	PROCESSING:
		CASE THIS^.intersectIterator.iterate(execute := TRUE, object => iteratedObject) OF
		CNM_ReturnTypes.SingleExecutionState.BUSY:
			IF THIS^.getEqualObject(object := iteratedObject, foundObject => intersectObject) THEN
				IF (THIS^.intersectedTree^.insert(intersectObject) <> CNM_ReturnTypes.SingleExecutionResult.ERROR) THEN
					insertOperationsThisCycle := insertOperationsThisCycle + log2(THIS^.intersectedTree^.size);
				ELSE
					cycleManager.proceedWith(ERROR);
					CONTINUE;
				END_IF
			END_IF
			insertOperationsThisCycle := insertOperationsThisCycle + log2(THIS^.size);
		CNM_ReturnTypes.SingleExecutionState.ERROR:
			cycleManager.proceedWith(ERROR);
			CONTINUE;
		CNM_ReturnTypes.SingleExecutionState.SUCCESS:
			THIS^.clear();
			THIS^.root := THIS^.intersectedTree^.root;
			THIS^.size := THIS^.intersectedTree^.size;
			THIS^.intersectedTree^.root := 0;
			THIS^.intersectedTree^.destruct();
			THIS^.intersectedTree := 0;
			THIS^.intersectIterator.destruct();
			THIS^.intersectIterator := 0;
			cycleManager.proceedWith(SUCCESS);
			CONTINUE;
		END_CASE
	
	ERROR:
		THIS^.intersectIterator.destruct();
		THIS^.intersectIterator := 0;
		__DELETE(THIS^.intersectedTree);
		THIS^.intersectedTree := 0;
	END_CASE	
UNTIL
	(insertOperationsThisCycle >= THIS^.maxCycleCompares) OR_ELSE
	(cycleManager.state <> CNM_ReturnTypes.SingleExecutionState.BUSY)
END_REPEAT

intersect := cycleManager.state;
END_METHOD


(*

## Short summary

This method returns the next object in the iteration and returns an execution state.

.. <legal notes>

legal notes
=================
| SPDX-FileCopyrightText: © 2022 ekvip automation GmbH <info@ekvip.de>
| SPDX-License-Identifier: Apache-2.0
| For details check: Apache-2.0_

.. _Apache-2.0: https://www.apache.org/licenses/LICENSE-2.0

.. </legal notes>


**Return:** ``SUCCESS``: if last object from collection was returned,
	``ABORTED``: execute has a falling edge during iterate,
	``BUSY``: When iterate had rising edge on execute and not all objects had been returned yet
	``IDLE``: iterate not in progress, execute is false and iterate reseted 
	
*)

METHOD PROTECTED iterate :CNM_ReturnTypes.SingleExecutionState
VAR_INPUT
	execute					:BOOL;
END_VAR
VAR_OUTPUT
	object					:CNM_AbstractObject.IObject;
END_VAR
VAR_INST
	currentNode				:CNM_CollectionInterfaces.IBinaryTreeNode;
	stacktop				:__XWORD := 0;
	cycleManager	:CNM_CycleManager.SimpleCycleManager;
	lastTreeVersion :__XWORD;
END_VAR
VAR 
	stacksize 				:UDINT;
END_VAR
VAR CONSTANT 
	INIT :DINT := CNM_ReturnTypes.DefaultSteps.STEP.INIT;
	ITERATING :DINT := INIT + 1;
	SUCCESS :DINT := CNM_ReturnTypes.DefaultSteps.STEP.SUCCESS;
	ERROR :DINT := CNM_ReturnTypes.DefaultSteps.STEP.ERROR;
	OBJECT_NOT_REFERENCED	:__XWORD := 0;
END_VAR
cycleManager(execute := execute);
CASE cycleManager.step.current OF
INIT:
	cycleManager.configuration.sequence.requireSuccessStep := FALSE;
	stacksize := THIS^.treeHeight;
	object := OBJECT_NOT_REFERENCED;
	lastTreeVersion := THIS^.changesToCollection;
	__DELETE(THIS^.nodestack);
	stacktop := 0;
	THIS^.nodestack := __NEW(__XWORD, stacksize);
	currentNode := THIS^.getSmallestNode(startNode:=THIS^.rootNode,nodebuffer := THIS^.nodestack,bufferindex := stacktop);
	IF THIS^.isObjectValid(currentNode) THEN
		object := currentNode.object;
		THIS^.getInorderSuccessor(
          nodebuffer := THIS^.nodestack, 
          bufferindex := stacktop, 
          successor => currentNode
        );
	END_IF
	cycleManager.proceedWith(
		step := SEL((THIS^.size > 0), SUCCESS, ITERATING)
	);
	
ITERATING:
	IF THIS^.changesToCollection <> lastTreeVersion THEN
		cycleManager.proceedWith(ERROR);
		iterate := CNM_ReturnTypes.SingleExecutionState.ERROR;
		RETURN;
	END_IF
	IF THIS^.isObjectValid(currentNode) THEN
		object := currentNode.object;
		THIS^.getInorderSuccessor(
          nodebuffer := THIS^.nodestack, 
          bufferindex := stacktop, 
          successor => currentNode
        );
	ELSE
		__DELETE(THIS^.nodestack);
		cycleManager.proceedWith(SUCCESS);
	END_IF
END_CASE

iterate := cycleManager.state;
END_METHOD

(*

## Short summary

This property defines the maximum amount of compares that should be done per Cycle. Is optional as default should be set by class.
Passing zero resets to class specific default.

.. <legal notes>

legal notes
=================
| SPDX-FileCopyrightText: © 2022 ekvip automation GmbH <info@ekvip.de>
| SPDX-License-Identifier: Apache-2.0
| For details check: Apache-2.0_

.. _Apache-2.0: https://www.apache.org/licenses/LICENSE-2.0

.. </legal notes>

*)

PROPERTY maxCycleCompares : UDINT
GET
maxCycleCompares := THIS^.upperCompareBound;
END_GET
SET
THIS^.upperCompareBound := SEL(
	maxCycleCompares = 0,
	maxCycleCompares,
	GeneralParameters.DEFAULT_OPERATIONS_PER_CYCLE
);
END_SET
END_PROPERTY

(*

## Short summary

overwrites the content of this set with the union of this set and the given set
Set union: Combination of all elements from two sets.

**Example:**
Set A = {2, 3, 1, 4}
Set B = {3, 5, 6, 4}

Union of A and B: {1, 2, 3, 4, 5, 6}

.. <legal notes>

legal notes
=================
| SPDX-FileCopyrightText: © 2022 ekvip automation GmbH <info@ekvip.de>
| SPDX-License-Identifier: Apache-2.0
| For details check: Apache-2.0_

.. _Apache-2.0: https://www.apache.org/licenses/LICENSE-2.0

.. </legal notes>


**Return:** ``SUCCESS``: if merge completed, 
	``ABORTED``: execute has a falling edge during merge,
	``BUSY``: merge is in Progress
	``ERROR``: the passed collection where not valid / contained invalid Elements
	``IDLE``: Currently no merge in progress

*)

METHOD INTERNAL merge :CNM_ReturnTypes.SingleExecutionState
VAR_INPUT
	(*foreign set to merge with*)
	set :CNM_CollectionInterfaces.ISet;
	(*If merge should be processed*)
	execute		:BOOL;
END_VAR
VAR
	object		 	:CNM_AbstractObject.IObject;
	iterateState	:CNM_ReturnTypes.SingleExecutionState;
END_VAR
merge := THIS^.insertCollection(
	collection := set,
	execute := execute);
END_METHOD

(*

## Short summary

recursiv insert function, tries to insert in the Tree and if not on right position call itself again on a subtree, on way out of recursin (re)balance tree

.. <legal notes>

legal notes
=================
| SPDX-FileCopyrightText: © 2022 ekvip automation GmbH <info@ekvip.de>
| SPDX-License-Identifier: Apache-2.0
| For details check: Apache-2.0_

.. _Apache-2.0: https://www.apache.org/licenses/LICENSE-2.0

.. </legal notes>


**Return:** the node that is the new root of the subtree for that the recursiv method is called

*)

METHOD PROTECTED recursivInsert :CNM_CollectionInterfaces.IBalancedBinarySearchTreeNode
VAR_INPUT
	(*the object that shoul be inserted*)
	object 						:CNM_AbstractObject.IObject;
	(*the root of the tree we try to insert in*)
	elem 						:CNM_CollectionInterfaces.IBalancedBinarySearchTreeNode;
END_VAR
VAR_IN_OUT
	(*is changed to false when insert was successful*)
	heightNotChanged 			:BOOL;
END_VAR
VAR 
	rightChild 					:CNM_CollectionInterfaces.IBalancedBinarySearchTreeNode;
	binaryRightChild 			:CNM_CollectionInterfaces.IBinaryTreeNode;
	binaryLeftChild 			:CNM_CollectionInterfaces.IBinaryTreeNode;
	leftChild		  			:CNM_CollectionInterfaces.IBalancedBinarySearchTreeNode;
END_VAR
VAR_OUTPUT
	(*SUCCESS if node could be inserted, ERROR if object already in the tree, ABORTED if object was null or empty node found*)
	insertResult 				:CNM_ReturnTypes.SingleExecutionResult;
END_VAR
VAR CONSTANT
	OBJECT_IS_NOT_REFERENCED	:__XWORD := 0; 
END_VAR
IF THIS^.isObjectNull(elem) AND NOT THIS^.isObjectNull(object) THEN
	IF (THIS^.collectionFactory.getNewBBSTreeNode(object := object, node => recursivInsert) <> CNM_ReturnTypes.SingleExecutionResult.SUCCESS) THEN
		insertResult := CNM_ReturnTypes.SingleExecutionResult.ERROR;
	ELSE
		insertResult := CNM_ReturnTypes.SingleExecutionResult.SUCCESS;
	END_IF
	RETURN;
ELSIF  THIS^.isObjectNull(object) OR_ELSE THIS^.isObjectNull(elem.object) THEN
	insertResult := CNM_ReturnTypes.SingleExecutionResult.ABORTED;
	RETURN;
END_IF
	

CASE THIS^.compareNodes(object, elem.object) OF
 	CNM_ReturnTypes.ComparationResult.EQUAL:
		recursivInsert := elem;
		insertResult := CNM_ReturnTypes.SingleExecutionResult.ABORTED;
		RETURN;
 	CNM_ReturnTypes.ComparationResult.SMALLER: 
		IF (THIS^.isObjectNull(elem.leftChild)) THEN
			IF (THIS^.collectionFactory.getNewBBSTreeNode(object := object, node => leftChild) = CNM_ReturnTypes.SingleExecutionResult.SUCCESS) THEN
				__QUERYINTERFACE(leftChild, binaryLeftChild);
				elem.leftChild := binaryLeftChild;
				heightNotChanged := FALSE;
				insertResult := CNM_ReturnTypes.SingleExecutionResult.SUCCESS;
			ELSE
				insertResult := CNM_ReturnTypes.SingleExecutionResult.ERROR;
			END_IF
		ELSE
			__QUERYINTERFACE(elem.leftChild, leftChild);
			leftChild := THIS^.recursivInsert(object := object, elem := leftChild, heightNotChanged := heightNotChanged, insertResult => insertResult);	
			__QUERYINTERFACE(leftChild,binaryLeftChild);
			elem.leftChild := binaryLeftChild;
		END_IF
		recursivInsert := THIS^.checkRightRotation(elem:=elem,heightNotChanged:=heightNotChanged, removing := FALSE);
		RETURN;
	CNM_ReturnTypes.ComparationResult.Greater:
		IF THIS^.isObjectNull(elem.rightChild) THEN 
			IF (THIS^.collectionFactory.getNewBBSTreeNode(object := object, node => rightChild) = CNM_ReturnTypes.SingleExecutionResult.SUCCESS) THEN
				__QUERYINTERFACE(rightChild,binaryRightChild);
				elem.rightChild := binaryRightChild;
				heightNotChanged := FALSE;
				insertResult := CNM_ReturnTypes.SingleExecutionResult.SUCCESS;
			ELSE
				insertResult := CNM_ReturnTypes.SingleExecutionResult.ERROR;
			END_IF
		ELSE
			__QUERYINTERFACE(elem.rightChild,rightChild);
			rightChild := THIS^.recursivInsert(object:=object,elem:=rightChild,heightNotChanged:=heightNotChanged,insertResult=>insertResult);
			__QUERYINTERFACE(rightChild,binaryRightChild);
			elem.rightChild := binaryRightChild;	
		END_IF
		recursivInsert := THIS^.checkLeftRotation(elem:=elem,heightNotChanged:=heightNotChanged,removing := FALSE);
		RETURN;
END_CASE;
END_METHOD

(*

## Short summary

recursiv remove an element tries to remove element from tree, if not possible calls itself on subtree, on way out of recursin (re)balance tree

.. <legal notes>

legal notes
=================
| SPDX-FileCopyrightText: © 2022 ekvip automation GmbH <info@ekvip.de>
| SPDX-License-Identifier: Apache-2.0
| For details check: Apache-2.0_

.. _Apache-2.0: https://www.apache.org/licenses/LICENSE-2.0

.. </legal notes>


**Return:** the node that is the new root of the subtree for that the recursiv method is called

*)

METHOD PROTECTED recursivRemove :CNM_CollectionInterfaces.IBalancedBinarySearchTreeNode
VAR_INPUT
	(*The object that should be removed*)
	object 						:CNM_AbstractObject.IObject;
	(*The root of the tree we try to delete the object from *)
	elem 						:CNM_CollectionInterfaces.IBalancedBinarySearchTreeNode;
END_VAR
VAR_IN_OUT
	(*changed to false when node is removed*)
	heightNotChanged 			:BOOL;
END_VAR
VAR 
	leftChild					:CNM_CollectionInterfaces.IBalancedBinarySearchTreeNode;
	binaryLeftChild 			:CNM_CollectionInterfaces.IBinaryTreeNode;
	binaryRightChild 			:CNM_CollectionInterfaces.IBinaryTreeNode;
	rightChild 					:CNM_CollectionInterfaces.IBalancedBinarySearchTreeNode;
	testrightChild 				:CNM_CollectionInterfaces.IBinaryTreeNode;
END_VAR
VAR_OUTPUT
	(*SUCCESS, if remove was successful*)
	removeResult 				:CNM_ReturnTypes.SingleExecutionResult;
END_VAR
VAR CONSTANT
	OBJECT_IS_NOT_REFERENCED	:__XWORD := 0;
END_VAR
IF THIS^.isObjectNull(elem) THEN
	recursivRemove := OBJECT_IS_NOT_REFERENCED;
	removeResult := CNM_ReturnTypes.SingleExecutionResult.ABORTED;
	RETURN;
ELSIF THIS^.isObjectNull(object) OR_ELSE THIS^.isObjectNull(elem.object) THEN
	removeResult := CNM_ReturnTypes.SingleExecutionResult.ERROR;
	RETURN;
END_IF;

CASE THIS^.compareNodes(object,elem.object) OF
	CNM_AbstractObject.CNM_ReturnTypes.ComparationResult.SMALLER:
		__QUERYINTERFACE(elem.leftChild,leftChild);
		leftChild := THIS^.recursivRemove(object:=object,elem:=leftChild, heightNotChanged := heightNotChanged,removeResult=>removeResult);
		__QUERYINTERFACE(leftChild,binaryLeftChild);
		elem.leftChild := binaryLeftChild;
		recursivRemove := checkLeftRotation(elem := elem, heightNotChanged := heightNotChanged,removing := TRUE);
		RETURN;
	CNM_AbstractObject.CNM_ReturnTypes.ComparationResult.GREATER:
		__QUERYINTERFACE(elem.rightChild,rightChild);
		rightChild := THIS^.recursivRemove(object := object, elem := rightChild, heightNotChanged := heightNotChanged,removeResult=>removeResult);
		__QUERYINTERFACE(rightChild,binaryRightChild);
		elem.rightChild := binaryRightChild;
		recursivRemove := checkRightRotation(elem := elem, heightNotChanged := heightNotChanged,removing := TRUE);
		RETURN;
	CNM_AbstractObject.CNM_ReturnTypes.ComparationResult.EQUAL:
		IF THIS^.isObjectNull(elem.leftChild) THEN
			heightNotChanged := FALSE;
			__QUERYINTERFACE(elem.rightChild,recursivRemove);
			
		ELSIF THIS^.isObjectNull(elem.rightChild) THEN
			heightNotChanged:=FALSE;
			__QUERYINTERFACE(elem.leftChild,recursivRemove);
		ELSE
			recursivRemove := searchSuccessor(elem:=elem,heightNotChanged:=heightNotChanged);
			recursivRemove.balance := elem.balance;
			recursivRemove.leftChild := elem.leftChild;
			recursivRemove.rightChild := elem.rightChild;
			recursivRemove := checkRightRotation(elem := recursivRemove,heightNotChanged:=heightNotChanged,removing := TRUE);
		END_IF
		removeResult := CNM_ReturnTypes.SingleExecutionResult.SUCCESS;
		elem.leftChild := OBJECT_IS_NOT_REFERENCED;
		elem.rightChild := OBJECT_IS_NOT_REFERENCED;
		elem.destruct();
		RETURN;
END_CASE
END_METHOD

(*

## Short summary

gets the successor of a node and removes it from the tree so it can be inserted at another place (used when remove) and rebalances tree

.. <legal notes>

legal notes
=================
| SPDX-FileCopyrightText: © 2022 ekvip automation GmbH <info@ekvip.de>
| SPDX-License-Identifier: Apache-2.0
| For details check: Apache-2.0_

.. _Apache-2.0: https://www.apache.org/licenses/LICENSE-2.0

.. </legal notes>


**Return:** The successor node of the elem node

*)

METHOD PROTECTED recursivSearchSuccessor :CNM_CollectionInterfaces.IBalancedBinarySearchTreeNode
VAR_INPUT
	(*the element a successor should be searched for*)
	elem 				:CNM_CollectionInterfaces.IBalancedBinarySearchTreeNode;
END_VAR
VAR_IN_OUT
	(*True if the successor was removed*)
	heightNotChanged 	:BOOL;
END_VAR
VAR_OUTPUT
	(*returns the new root, bc root can be changed bc of rotation*)
	newRoot				:CNM_CollectionInterfaces.IBalancedBinarySearchTreeNode;
END_VAR
VAR
	leftChild			:CNM_CollectionInterfaces.IBalancedBinarySearchTreeNode;
END_VAR
IF NOT THIS^.isObjectNull(elem.leftChild.leftChild) THEN
	__QUERYINTERFACE(elem.leftChild,leftChild);
	recursivSearchSuccessor := THIS^.recursivSearchSuccessor(elem:=leftChild,heightNotChanged := heightNotChanged,newRoot => newRoot);
	elem.leftChild := newRoot;
	newRoot := checkLeftRotation(elem:=elem,heightNotChanged:=heightNotChanged,removing:=TRUE);
	RETURN;
ELSE
	__QUERYINTERFACE(elem.leftChild,leftChild);
	recursivSearchSuccessor := leftChild;
	elem.leftChild := elem.leftChild.rightChild;
	newRoot := checkLeftRotation(elem:=elem,heightNotChanged:=heightNotChanged,removing:=TRUE);
	RETURN;
END_IF
END_METHOD


(*

## Short summary

Method to remove an object from the tree.

.. <legal notes>

legal notes
=================
| SPDX-FileCopyrightText: © 2022 ekvip automation GmbH <info@ekvip.de>
| SPDX-License-Identifier: Apache-2.0
| For details check: Apache-2.0_

.. _Apache-2.0: https://www.apache.org/licenses/LICENSE-2.0

.. </legal notes>


**Return:** ``SUCCESS``: if remove could be made
	``ABORTED``: if object wasn't in the tree
	``ERROR``: if object wasn't valid

*)

METHOD INTERNAL remove :CNM_ReturnTypes.SingleExecutionResult
VAR_INPUT
	(* The object that should be removed *)
	object				:CNM_AbstractObject.IObject;
END_VAR
VAR
	heightNotChanged	:BOOL := TRUE;
	newRootNode				:CNM_CollectionInterfaces.IBalancedBinarySearchTreeNode;
END_VAR
newRootNode := THIS^.recursivRemove(
	object:=object,
	elem:=THIS^.rootNode,
	heightNotChanged := heightNotChanged,
	removeResult=>remove
);
IF remove = CNM_ReturnTypes.SingleExecutionResult.SUCCESS THEN
	THIS^.decrementSize();
	THIS^.announceChange();
	THIS^.rootNode := newRootNode;
	RETURN;		
END_IF
END_METHOD

(*

## Short summary

performs a left rotation around a specified node and cares about the subtress and balance
 
.. <legal notes>

legal notes
=================
| SPDX-FileCopyrightText: © 2022 ekvip automation GmbH <info@ekvip.de>
| SPDX-License-Identifier: Apache-2.0
| For details check: Apache-2.0_

.. _Apache-2.0: https://www.apache.org/licenses/LICENSE-2.0

.. </legal notes>


**Return:** the new root that replaced the one that was used for rotation

*)

METHOD PROTECTED reorganizeLeftRotate :CNM_CollectionInterfaces.IBalancedBinarySearchTreeNode
VAR_INPUT
	(*The element around that should be rotatet*)
	elem				:CNM_CollectionInterfaces.IBalancedBinarySearchTreeNode;
	(*indicates if method was called in context of remove (then true) or in context of insert (then false) *)
	removing				:BOOL;
END_VAR
VAR_IN_OUT
	(*false if the height of the tree changed*)
	heightNotChanged 	:BOOL;
END_VAR
VAR 
	internLeftChild		:CNM_CollectionInterfaces.IBalancedBinarySearchTreeNode;
	internRightChild	:CNM_CollectionInterfaces.IBalancedBinarySearchTreeNode; 
END_VAR
__QUERYINTERFACE(elem.rightChild,internRightChild);

CASE internRightChild.balance OF
	CNM_CollectionInterfaces.TreeBalance.RIGHTDEEPER:
		elem := THIS^.rotateLeft(elem);
		__QUERYINTERFACE(elem.leftChild,internLeftChild);
		internLeftChild.balance := CNM_CollectionInterfaces.TreeBalance.EQUALDEEP;
		elem.balance := CNM_CollectionInterfaces.TreeBalance.EQUALDEEP;
		heightNotChanged := NOT removing;
		reorganizeLeftRotate := elem;
	CNM_CollectionInterfaces.TreeBalance.EQUALDEEP: 
		elem := THIS^.rotateLeft(elem);
		__QUERYINTERFACE(elem.leftChild,internLeftChild);
		internLeftChild.balance := CNM_CollectionInterfaces.TreeBalance.RIGHTDEEPER;
		elem.balance := CNM_CollectionInterfaces.TreeBalance.LEFTDEEPER;
		heightNotChanged := removing;
		reorganizeLeftRotate := elem;
	CNM_CollectionInterfaces.TreeBalance.LEFTDEEPER:
		elem.rightChild := THIS^.rotateRight(internRightChild);
		elem := THIS^.rotateLeft(elem);
		THIS^.adaptBalanceAfterDoubleRotation(elem:=elem);
		elem.balance := CNM_CollectionInterfaces.TreeBalance.EQUALDEEP;
		heightNotChanged := removing;
		reorganizeLeftRotate := elem;
END_CASE
END_METHOD

(*

## Short summary

rotates right around a specified node, and cares about subtrees and balance

.. <legal notes>

legal notes
=================
| SPDX-FileCopyrightText: © 2022 ekvip automation GmbH <info@ekvip.de>
| SPDX-License-Identifier: Apache-2.0
| For details check: Apache-2.0_

.. _Apache-2.0: https://www.apache.org/licenses/LICENSE-2.0

.. </legal notes>


**Return:** the node that replaced the node that was used to rotate around

*)

METHOD PROTECTED reorganizeRightRotate :CNM_CollectionInterfaces.IBalancedBinarySearchTreeNode
VAR_INPUT
	(*the node around the rotation should be performed*)
	elem 				:CNM_CollectionInterfaces.IBalancedBinarySearchTreeNode;
	(*indicates if method was called in context of remove (then true) or in context of insert (then false) *)
	removing 				:BOOL;
END_VAR
VAR_IN_OUT
	(*false if height changed, set to true when rotation rebalanced the tree*)
	heightNotChanged 	:BOOL;
END_VAR
VAR 
	leftChild 			:CNM_CollectionInterfaces.IBalancedBinarySearchTreeNode;
	rightChild 			:CNM_CollectionInterfaces.IBalancedBinarySearchTreeNode;
END_VAR
__QUERYINTERFACE(elem.leftChild,leftChild);
__QUERYINTERFACE(elem.rightChild, rightChild);

CASE leftChild.balance OF 
	CNM_CollectionInterfaces.TreeBalance.LEFTDEEPER: 
		elem := rotateRight(elem:=elem);
		__QUERYINTERFACE(elem.rightChild, rightChild);
		rightChild.balance := CNM_CollectionInterfaces.TreeBalance.EQUALDEEP;
		elem.balance := CNM_CollectionInterfaces.TreeBalance.EQUALDEEP;
		heightNotChanged := NOT removing;
		reorganizeRightRotate := elem;
		RETURN;
	CNM_CollectionInterfaces.TreeBalance.EQUALDEEP: 
		elem := rotateRight(elem:=elem);
		__QUERYINTERFACE(elem.rightChild, rightChild);
		rightChild.balance := CNM_CollectionInterfaces.TreeBalance.LEFTDEEPER;
		elem.balance := CNM_CollectionInterfaces.TreeBalance.RIGHTDEEPER;
		heightNotChanged := removing;
		reorganizeRightRotate := elem;
		RETURN;
	CNM_CollectionInterfaces.TreeBalance.RIGHTDEEPER:
		elem.leftChild := rotateLeft(elem:=leftChild);
		elem := rotateRight(elem:=elem);
		adaptBalanceAfterDoubleRotation(elem:=elem);
		elem.balance := CNM_CollectionInterfaces.TreeBalance.EQUALDEEP;
		heightNotChanged := NOT removing;
		reorganizeRightRotate := elem;
		RETURN;
		
END_CASE
END_METHOD

(*

## Short summary

This property points to the root of a tree

.. <legal notes>

legal notes
=================
| SPDX-FileCopyrightText: © 2022 ekvip automation GmbH <info@ekvip.de>
| SPDX-License-Identifier: Apache-2.0
| For details check: Apache-2.0_

.. _Apache-2.0: https://www.apache.org/licenses/LICENSE-2.0

.. </legal notes>

*)
PROPERTY INTERNAL root : CNM_CollectionInterfaces.IBalancedBinarySearchTreeNode
GET
root := THIS^.rootNode;
END_GET
SET
THIS^.rootNode := root;
END_SET
END_PROPERTY

(*

## Short summary

rotates a tree around a node

.. <legal notes>

legal notes
=================
| SPDX-FileCopyrightText: © 2022 ekvip automation GmbH <info@ekvip.de>
| SPDX-License-Identifier: Apache-2.0
| For details check: Apache-2.0_

.. _Apache-2.0: https://www.apache.org/licenses/LICENSE-2.0

.. </legal notes>


**Return:** the new root

*)

METHOD PROTECTED rotateLeft :CNM_CollectionInterfaces.IBalancedBinarySearchTreeNode
VAR_INPUT
	(*The element that sould be rotatet around*)
	elem	:CNM_CollectionInterfaces.IBalancedBinarySearchTreeNode;
END_VAR
VAR 
	newRoot	:CNM_CollectionInterfaces.IBalancedBinarySearchTreeNode;	
END_VAR
__QUERYINTERFACE(elem.rightChild, newRoot);
elem.rightChild := newRoot.leftChild;
newRoot.leftChild := elem;
rotateLeft := newRoot;
END_METHOD

(*

## Short summary

rotates right around a specified node, doesnt care about balance and stuff, this is done in method ``reorganizeRightRotate``

.. <legal notes>

legal notes
=================
| SPDX-FileCopyrightText: © 2022 ekvip automation GmbH <info@ekvip.de>
| SPDX-License-Identifier: Apache-2.0
| For details check: Apache-2.0_

.. _Apache-2.0: https://www.apache.org/licenses/LICENSE-2.0

.. </legal notes>


**Return:** the new root

*)

METHOD PROTECTED rotateRight :CNM_CollectionInterfaces.IBalancedBinarySearchTreeNode
VAR_INPUT
	(*the element that should be rotatet around*)
	elem	:CNM_CollectionInterfaces.IBalancedBinarySearchTreeNode;
END_VAR
VAR
	newRoot	:CNM_CollectionInterfaces.IBalancedBinarySearchTreeNode;
END_VAR
__QUERYINTERFACE(elem.leftChild,newRoot);
elem.leftChild := newRoot.rightChild;
newRoot.rightChild := elem;
rotateRight := newRoot;
END_METHOD

(*

## Short summary

searches a successor and removes it from the tree so it can be used to replace another (deleted) node

.. <legal notes>

legal notes
=================
| SPDX-FileCopyrightText: © 2022 ekvip automation GmbH <info@ekvip.de>
| SPDX-License-Identifier: Apache-2.0
| For details check: Apache-2.0_

.. _Apache-2.0: https://www.apache.org/licenses/LICENSE-2.0

.. </legal notes>


**Return:** The successor node

*)

METHOD PROTECTED searchSuccessor :CNM_CollectionInterfaces.IBalancedBinarySearchTreeNode
VAR_INPUT
	(*The element that the successor is searched from*)
	elem 				:CNM_CollectionInterfaces.IBalancedBinarySearchTreeNode;
END_VAR
VAR_IN_OUT
	(*True if operation did not change the height of the subtree / heightchange was handled*)
	heightNotChanged 	:BOOL;
END_VAR
VAR
	newRoot				:CNM_CollectionInterfaces.IBalancedBinarySearchTreeNode;
	rightChild			:CNM_CollectionInterfaces.IBalancedBinarySearchTreeNode;
END_VAR
__QUERYINTERFACE(elem.rightChild,rightChild);
IF THIS^.isObjectNull(elem.rightChild.leftChild) THEN
	searchSuccessor := rightChild;
	elem.rightChild := elem.rightChild.rightChild;
	heightNotChanged := FALSE;
	RETURN;
ELSE
	searchSuccessor := recursivSearchSuccessor(elem:=rightChild,heightNotChanged:=heightNotChanged,newRoot=>newRoot);
	elem.rightChild := newRoot;
	RETURN;
END_IF
END_METHOD

(*

## Short summary

This property returns a fluent interface to set operations, e.g. intersect() and subtract().

.. <legal notes>

legal notes
=================
| SPDX-FileCopyrightText: © 2025 ekvip automation GmbH <info@ekvip.de>
| SPDX-License-Identifier: Apache-2.0
| For details check: Apache-2.0_

.. _Apache-2.0: https://www.apache.org/licenses/LICENSE-2.0

.. </legal notes>

*)

PROPERTY set :CNM_CollectionInterfaces.ISetStrategy
GET
VAR_INST
	setExecutor :SetStrategyExecutor(THIS^);
END_VAR
set := setExecutor;
END_GET
END_PROPERTY

(*

## Short summary

Sets a comparator, that is used to compare two nodes of this tree.
Optional, if not set, object.compareTo will be used.

**Attention:**
	The comparator can only be set if the tree has at most one element.

**Attention:**
	Will be deep destructed within the deep destruct context of this class.

.. <legal notes>

legal notes
=================
| SPDX-FileCopyrightText: © 2022 ekvip automation GmbH <info@ekvip.de>
| SPDX-License-Identifier: Apache-2.0
| For details check: Apache-2.0_

.. _Apache-2.0: https://www.apache.org/licenses/LICENSE-2.0

.. </legal notes>


**Return:** ``SUCCESS``: new comparator was set
	``ABORTED``: tree already contained more than one object
	
*)

METHOD setNodeComparator :CNM_ReturnTypes.SingleExecutionResult
VAR_INPUT
	(*the comparator that should be used to compare two nodes*)
	nodeComparator	:CNM_AbstractObject.IComparator;
END_VAR
VAR CONSTANT
	MAXIMUM_SIZE_TO_SET_COMPARATOR :UDINT := 1;
END_VAR
IF THIS^.size > MAXIMUM_SIZE_TO_SET_COMPARATOR THEN
	setNodeComparator := CNM_ReturnTypes.SingleExecutionResult.ABORTED;
ELSE
	THIS^.nodeComparator := nodeComparator;
	setNodeComparator := CNM_ReturnTypes.SingleExecutionResult.SUCCESS;
END_IF
END_METHOD

(*

## Short summary

This property allows to change the collection size without using insert / remove etc.
Can be used for clone operations etc. should never be visible for the user.

.. <legal notes>

legal notes
=================
| SPDX-FileCopyrightText: © 2023 ekvip automation GmbH <info@ekvip.de>
| SPDX-License-Identifier: Apache-2.0
| For details check: Apache-2.0_

.. _Apache-2.0: https://www.apache.org/licenses/LICENSE-2.0

.. </legal notes>

*)

PROPERTY INTERNAL size :UDINT
SET
THIS^.collectionSize := size;
END_SET
END_PROPERTY

(*

## Short summary

overwrites the content of this set with the set difference of this set and the given set
Set difference: Elements present in one set but not in the other.

**Example:**
Set A = {2, 3, 1, 4}
Set B = {3, 5, 6, 4}

Set difference (A - B): {1, 2}
Set difference (B - A): {5, 6}

.. <legal notes>

legal notes
=================
| SPDX-FileCopyrightText: © 2025 ekvip automation GmbH <info@ekvip.de>
| SPDX-License-Identifier: Apache-2.0
| For details check: Apache-2.0_

.. _Apache-2.0: https://www.apache.org/licenses/LICENSE-2.0

.. </legal notes>


**Return:** ``SUCCESS``: if insert could made, error if object was already in the tree,
	``ABORTED``: execute has a falling edge during insert,
	``BUSY``: Insert is in Progress
	``ERROR``: the passed collection where not valid / contained invalid Elements
	``IDLE``: Currently no insert in progress

*)

METHOD INTERNAL subtract :CNM_ReturnTypes.SingleExecutionState
VAR_INPUT
	(*foreign set to construct substraction*)
	set 						:CNM_CollectionInterfaces.ISet;
	(*If substract should be processed*)
	execute						:BOOL;
END_VAR
VAR_INST
	cycleManager :CNM_CycleManager.SimpleCycleManager;
	changeIndex :__XWORD;
END_VAR
VAR
	object 						:CNM_AbstractObject.IObject;
	iterateState				:CNM_ReturnTypes.SingleExecutionState;
	insertOperationsThisCycle	:__XWORD;
END_VAR
VAR CONSTANT
	INIT :DINT := CNM_ReturnTypes.DefaultSteps.STEP.INIT;
	PROCESSING :DINT := INIT + 1;
	SUCCESS :DINT := CNM_ReturnTypes.DefaultSteps.STEP.SUCCESS;
	ERROR :DINT := CNM_ReturnTypes.DefaultSteps.STEP.ERROR;
END_VAR
IF THIS^.isObjectNull(set) THEN
	subtract := CNM_ReturnTypes.SingleExecutionState.ERROR;
	cycleManager.proceedWith(ERROR);
	RETURN;
END_IF
insertOperationsThisCycle := 0;
REPEAT
	cycleManager(execute := execute);
	CASE cycleManager.step.current OF
	INIT:
		cycleManager.configuration.sequence.requireSuccessStep := FALSE;
		IF ((THIS^.size = 0) OR_ELSE (set.size = 0)) THEN
			cycleManager.proceedWith(SUCCESS);
			subtract := CNM_ReturnTypes.SingleExecutionState.SUCCESS;
			RETURN;
		END_IF
		IF THIS^.isObjectValid(THIS^.subtractIterator) THEN
			THIS^.subtractIterator.destruct();
		END_IF
		IF (set.createNewIterator(iterator => THIS^.subtractIterator) <> CNM_ReturnTypes.SingleExecutionResult.SUCCESS) 
		THEN
			cycleManager.proceedWith(ERROR);
			subtract := CNM_ReturnTypes.SingleExecutionState.ERROR;
			RETURN;
		END_IF
		THIS^.subtractIterator.iterate(execute := FALSE);	
		changeIndex := THIS^.changesToCollection;
		cycleManager.proceed();
		
	PROCESSING:
		IF (changeIndex <> THIS^.changesToCollection) THEN
			cycleManager.proceedWith(ERROR);
			subtract := CNM_ReturnTypes.SingleExecutionState.ERROR;
			RETURN;
		END_IF
		WHILE (( iterateState := THIS^.subtractIterator.iterate(execute := TRUE, object => object)) = CNM_ReturnTypes.SingleExecutionState.BUSY) DO
			CASE THIS^.remove(object) OF
			CNM_ReturnTypes.SingleExecutionResult.ERROR:
				subtract := CNM_ReturnTypes.SingleExecutionState.ERROR;
				cycleManager.proceedWith(ERROR);
				RETURN;
			END_CASE
			insertOperationsThisCycle := (insertOperationsThisCycle + THIS^.treeHeight);
			IF (insertOperationsThisCycle >= THIS^.maxCycleCompares) THEN
				EXIT;
			END_IF
		END_WHILE
		
		CASE iterateState OF
		CNM_ReturnTypes.SingleExecutionState.SUCCESS:
			THIS^.subtractIterator.destruct();
			cycleManager.proceedWith(SUCCESS);
		CNM_ReturnTypes.SingleExecutionState.ERROR:
			THIS^.subtractIterator.destruct();
			cycleManager.proceedWith(ERROR);
		END_CASE
	
	END_CASE
UNTIL
	(insertOperationsThisCycle >= THIS^.maxCycleCompares) OR_ELSE
	(cycleManager.state <> CNM_ReturnTypes.SingleExecutionState.BUSY)
END_REPEAT
subtract := cycleManager.state;
END_METHOD

(*

## Short summary

This property returns a fluent interface to tree operations, e.g. insert() and remove().

.. <legal notes>

legal notes
=================
| SPDX-FileCopyrightText: © 2025 ekvip automation GmbH <info@ekvip.de>
| SPDX-License-Identifier: Apache-2.0
| For details check: Apache-2.0_

.. _Apache-2.0: https://www.apache.org/licenses/LICENSE-2.0

.. </legal notes>

*)

PROPERTY tree : CNM_CollectionInterfaces.ITreeStrategy
GET
VAR_INST
	treeExecutor :TreeStrategyExecutor(THIS^);
END_VAR
tree := treeExecutor;
END_GET
END_PROPERTY

(*

## Short summary


Function to calculate the height of a tree, as its a balanced binary tree, is defined as 
height := log\ :sub:`2`\(Nodeamount) (Truncated)
log\ :sub:`2`\(x) := log(x)/log(2)

.. <legal notes>

legal notes
=================
| SPDX-FileCopyrightText: © 2022 ekvip automation GmbH <info@ekvip.de>
| SPDX-License-Identifier: Apache-2.0
| For details check: Apache-2.0_

.. _Apache-2.0: https://www.apache.org/licenses/LICENSE-2.0

.. </legal notes>

*)

PROPERTY PROTECTED treeHeight : USINT
GET
(*

## Short summary

Function to calculate the height of a tree, as its a balanced binary tree, is defined as 
height := log\ :sub:`2`\(Nodeamount) (Truncated)
log\ :sub:`2`\(x) := log(x)/log(2)

.. <legal notes>

legal notes
=================
| SPDX-FileCopyrightText: © 2022 ekvip automation GmbH <info@ekvip.de>
| SPDX-License-Identifier: Apache-2.0
| For details check: Apache-2.0_

.. _Apache-2.0: https://www.apache.org/licenses/LICENSE-2.0

.. </legal notes>

*)
VAR
END_VAR
treeHeight := log2(THIS^.size);
END_GET
END_PROPERTY

END_FUNCTION_BLOCK

// ---- BinaryTree/BBSTIterator/classes/InorderBbstIterator.TcPOU
(*

## Short summary

This class implements in order iteration strategy (sorted) for balanced binary search trees.

.. <legal notes>

legal notes
=================
| SPDX-FileCopyrightText: © 2025 ekvip automation GmbH <info@ekvip.de>
| SPDX-License-Identifier: Apache-2.0
| For details check: Apache-2.0_

.. _Apache-2.0: https://www.apache.org/licenses/LICENSE-2.0

.. </legal notes>

*)

{attribute 'enable_dynamic_creation'}
FUNCTION_BLOCK InorderBbstIterator EXTENDS AbstractBalancedBinarySearchTreeIterator

PROPERTY className :CNM_AbstractObject.ClassName
GET
className := 'CNM_Collections.InorderBBSTIterator';
END_GET
END_PROPERTY

(*

## Short summary

Searches the smallest childnode starting with the given node.
All visited nodes, will be added to the nodelist. This includes the smallest node as well.
 
.. <legal notes>

legal notes
=================
| SPDX-FileCopyrightText: © 2025 ekvip automation GmbH <info@ekvip.de>
| SPDX-License-Identifier: Apache-2.0
| For details check: Apache-2.0_

.. _Apache-2.0: https://www.apache.org/licenses/LICENSE-2.0

.. </legal notes>


**Return:** the successor node if found, or null if no successor exists

*)

METHOD PROTECTED FINAL fillNodeListUntilLeftMost
VAR_INPUT
	startNode	:CNM_CollectionInterfaces.IBinaryTreeNode;
END_VAR
VAR
	currentNode :CNM_CollectionInterfaces.IBinaryTreeNode;
END_VAR
VAR CONSTANT 
	OBJECT_NOT_REFERENCED	:__XWORD := 0;
END_VAR
RETURN(THIS^.isObjectNull(startNode));
currentNode := startNode;
WHILE(THIS^.isObjectValid(currentNode)) DO
	THIS^.nodeList.append(currentNode);
	currentNode := currentNode.leftChild;
END_WHILE
END_METHOD

(*

## Short summary

Gets the next node that iterate should process.

.. <legal notes>

legal notes
=================
| SPDX-FileCopyrightText: © 2022 ekvip automation GmbH <info@ekvip.de>
| SPDX-License-Identifier: Apache-2.0
| For details check: Apache-2.0_

.. _Apache-2.0: https://www.apache.org/licenses/LICENSE-2.0

.. </legal notes>


**Return:** ``TRUE`` a valid node existed, ``FALSE`` no node for iteration existed

*)

METHOD PROTECTED getNextTreeNode :BOOL
VAR_OUTPUT
	node	:CNM_CollectionInterfaces.IBinaryTreeNode;
END_VAR
VAR
	tmpObject	:CNM_AbstractObject.IObject;
END_VAR
tmpObject := THIS^.nodeList.pop();
__QUERYINTERFACE(tmpObject, node);
getNextTreeNode := THIS^.isObjectValid(node);
END_METHOD

(*

## Short summary

This method is called to retrive the first node of the iteration.
Might have sideeffects, like changes to THIS^.nodelist.

.. <legal notes>

legal notes
=================
| SPDX-FileCopyrightText: © 2022 ekvip automation GmbH <info@ekvip.de>
| SPDX-License-Identifier: Apache-2.0
| For details check: Apache-2.0_

.. _Apache-2.0: https://www.apache.org/licenses/LICENSE-2.0

.. </legal notes>



*)

METHOD PROTECTED getStartNode : CNM_CollectionInterfaces.IBinaryTreeNode
THIS^.fillNodeListUntilLeftMost(THIS^.root);
__QUERYINTERFACE(THIS^.nodeList.pop(), getStartNode);
END_METHOD

(*

## Short summary

This method appends (if they exists) the left and right child of the node to the nodelist.

.. <legal notes>

legal notes
=================
| SPDX-FileCopyrightText: © 2022 ekvip automation GmbH <info@ekvip.de>
| SPDX-License-Identifier: Apache-2.0
| For details check: Apache-2.0_

.. _Apache-2.0: https://www.apache.org/licenses/LICENSE-2.0

.. </legal notes>



*)

METHOD PROTECTED processNode
VAR_INPUT
	nodeToProcess	: CNM_CollectionInterfaces.IBinaryTreeNode;
END_VAR
THIS^.fillNodeListUntilLeftMost(nodeToProcess.rightChild);
END_METHOD

END_FUNCTION_BLOCK

// ---- BinaryTree/BBSTIterator/classes/AbstractBalancedBinarySearchTreeIterator.TcPOU
(*

## Short summary

This class provides the basic methods and functionalities for Balanced Binary Tree iterators.

.. <legal notes>

legal notes
=================
| SPDX-FileCopyrightText: © 2024 ekvip automation GmbH <info@ekvip.de>
| SPDX-License-Identifier: Apache-2.0
| For details check: Apache-2.0_

.. _Apache-2.0: https://www.apache.org/licenses/LICENSE-2.0

.. </legal notes>

*)

FUNCTION_BLOCK ABSTRACT AbstractBalancedBinarySearchTreeIterator EXTENDS AbstractIterator IMPLEMENTS IBBSTIterator
VAR	
	{attribute 'hide'}
	tree 		:REFERENCE TO BalancedBinarySearchTree;
	nodeList 	:LinkedList();
	currentNode :CNM_CollectionInterfaces.IBinaryTreeNode;
END_VAR

(*

## Short summary

This method attaches an binary balances search tree to the iterator.

.. <legal notes>

legal notes
=================
| SPDX-FileCopyrightText: © 2022 ekvip automation GmbH <info@ekvip.de>
| SPDX-License-Identifier: Apache-2.0
| For details check: Apache-2.0_

.. _Apache-2.0: https://www.apache.org/licenses/LICENSE-2.0

.. </legal notes>


**Return:** ``CNM_ReturnTypes.SingleExecutionResult.SUCCESS``: the tree could be attached to the iterator
	``CNM_ReturnTypes.SingleExecutionResult.ERROR``: the passed tree was not valid

*)

METHOD attachTree
VAR_INPUT
	tree : REFERENCE TO BalancedBinarySearchTree;
END_VAR
THIS^.tree REF= tree;
THIS^.reset();
END_METHOD

PROPERTY PROTECTED changes : __XWORD
GET
changes := THIS^.tree.changesToCollection;
END_GET
END_PROPERTY

(*

## Short summary

Mark the object as deleted, as it staiys in the memory.

.. <legal notes>

legal notes
=================
| SPDX-FileCopyrightText: © 2022 ekvip automation GmbH <info@ekvip.de>
| SPDX-License-Identifier: Apache-2.0
| For details check: Apache-2.0_

.. _Apache-2.0: https://www.apache.org/licenses/LICENSE-2.0

.. </legal notes>

*)
METHOD FB_Exit : BOOL
VAR_INPUT
	(* TRUE: the exit method is called in order to leave the instance which will be copied afterwards (online change).*)
	bInCopyCode	: BOOL;
END_VAR
IF THIS^.isObjectValid(THIS^.nodeList) THEN
	THIS^.nodeList.clear();
END_IF
END_METHOD

(*

## Short summary

The constructor ``FB_init`` is needed to create an unique hash code.
The hash code is a pseudo random number create with a [xorshift](https://en.wikipedia.org/wiki/Xorshift) algorithm.
It can be overwritten on derivations, because it will be called implicit, ``SUPER^.FB_init()`` is not required.
For more information check: [Behavoir with derived function blocks](https://infosys.beckhoff.com/content/1033/tc3_plc_intro/5482088715.html?id=6983869892358031022).

.. <legal notes>

legal notes
=================
| SPDX-FileCopyrightText: © 2022 ekvip automation GmbH <info@ekvip.de>
| SPDX-License-Identifier: Apache-2.0
| For details check: Apache-2.0_

.. _Apache-2.0: https://www.apache.org/licenses/LICENSE-2.0

.. </legal notes>



*)
METHOD FB_init : BOOL
VAR_INPUT
	(* if TRUE, the retain variables are initialized (warm start / cold start)*)
	bInitRetains	: BOOL;
	(* if TRUE, the instance afterwards gets moved into the copy code (online change) *)
	bInCopyCode	: BOOL;
	(*The tree that should be iterated, can be 0*)
	tree	:REFERENCE TO BalancedBinarySearchTree;	
END_VAR
THIS^.tree REF= tree;
IF THIS^.isObjectValid(tree) THEN
	THIS^.nodeList.append(THIS^.root);
	THIS^.currentNode := THIS^.root;	
END_IF
END_METHOD

(*

## Short summary

Gets the next Node that iterate should process.

.. <legal notes>

legal notes
=================
| SPDX-FileCopyrightText: © 2022 ekvip automation GmbH <info@ekvip.de>
| SPDX-License-Identifier: Apache-2.0
| For details check: Apache-2.0_

.. _Apache-2.0: https://www.apache.org/licenses/LICENSE-2.0

.. </legal notes>


**Return:** ``TRUE`` a valid node existed, ``FALSE`` no node for iteration existed

*)

METHOD PROTECTED ABSTRACT getNextTreeNode :BOOL
VAR_OUTPUT
	node :CNM_CollectionInterfaces.IBinaryTreeNode;
END_VAR
END_METHOD

(*

## Short summary

This method is called to retrive the first node of the iteration.
Might have sideeffects, like changes to THIS^.nodelist.

.. <legal notes>

legal notes
=================
| SPDX-FileCopyrightText: © 2022 ekvip automation GmbH <info@ekvip.de>
| SPDX-License-Identifier: Apache-2.0
| For details check: Apache-2.0_

.. _Apache-2.0: https://www.apache.org/licenses/LICENSE-2.0

.. </legal notes>



*)

METHOD PROTECTED getStartNode : CNM_CollectionInterfaces.IBinaryTreeNode
getStartNode := THIS^.root;
END_METHOD

(*

## Short summary

This method returns if there exists another element to iterate to.

**Example:**
```
WHILE(iterator.hasNext())DO
	iterator.getNext().foo();
END_WHILE
```

.. <legal notes>

legal notes
=================
| SPDX-FileCopyrightText: © 2022 ekvip automation GmbH <info@ekvip.de>
| SPDX-License-Identifier: Apache-2.0
| For details check: Apache-2.0_

.. _Apache-2.0: https://www.apache.org/licenses/LICENSE-2.0

.. </legal notes>


**Return:** ``TRUE``: Iterator has a next object that can be fetched with getNext()
	``FALSE``: Iterator finished

*)
METHOD hasNext : BOOL
hasNext := THIS^.nodeList.hasElement;
END_METHOD

(*

## Short summary

This method returns the next object in the iteration and returns an execution state.
**Example:**
You have a list: 1 2 3
the first iterate call will return CNM_ReturnTypes.BUSY and object = 1
the second iterate call will return CNM_ReturnTypes.BUSY and object = 2
the third iterate call will return CNM_ReturnTypes.BUSY and object = 3
the forth iterate call will return CNM_ReturnTypes.SUCCESS and object = NULL

.. <legal notes>

legal notes
=================
| SPDX-FileCopyrightText: © 2022 ekvip automation GmbH <info@ekvip.de>
| SPDX-License-Identifier: Apache-2.0
| For details check: Apache-2.0_

.. _Apache-2.0: https://www.apache.org/licenses/LICENSE-2.0

.. </legal notes>


**Return:** ``SingleExecutionState.SUCCESS``: Iteration finished, no new elements, returned NULL object
    ``SingleExecutionState.ERROR``: error during iteration
    ``SingleExecutionState.ABORT``: iteration aborted
    ``SingleExecutionState.BUSY``: returned an element and iteration in progress	
    ``SingleExecutionState.IDLE``: ready for iteration

*)
METHOD iterate : CNM_ReturnTypes.SingleExecutionState
VAR_INPUT
	execute	: BOOL;
END_VAR
VAR_OUTPUT
	object :CNM_AbstractObject.IObject;
END_VAR
VAR
	tmp : POINTER TO CNM_AbstractObject.Object;
END_VAR
VAR_INST
	cycleManager :CNM_CycleManager.SimpleCycleManager;
	lastExecute :BOOL;
	lastChangeVersion :__XWORD;
END_VAR
VAR CONSTANT
	INIT :DINT := CNM_ReturnTypes.DefaultSteps.STEP.INIT;
	ITERATING :DINT := INIT + 1;
	ERROR :DINT := CNM_ReturnTypes.DefaultSteps.STEP.ERROR;
	SUCCESS :DINT := CNM_ReturnTypes.DefaultSteps.STEP.SUCCESS;
	NULL: __XWORD := 0;
END_VAR
iterate := CNM_ReturnTypes.SingleExecutionState.ERROR;
RETURN (NOT THIS^.isObjectValid(THIS^.tree));
cycleManager(execute := execute);
CASE cycleManager.step.current OF
INIT:
	cycleManager.configuration.sequence.requireSuccessStep := FALSE;
	lastChangeVersion := THIS^.changes;
	THIS^.nodeList.clear();
	THIS^.currentNode := THIS^.getStartNode();
	IF THIS^.isObjectValid(THIS^.currentNode) THEN
		THIS^.processStartNode(THIS^.currentNode);
		THIS^.currentObject := THIS^.currentNode.object;
	ELSE
		THIS^.currentObject := 0;
	END_IF 
	
	cycleManager.proceedWith(
		step := SEL(
			THIS^.hasNext(),
			SUCCESS,
			ITERATING
		)
	);
ITERATING:
	IF lastChangeVersion <> THIS^.changes THEN
		iterate := CNM_ReturnTypes.SingleExecutionState.ERROR;
		cycleManager.proceedWith(ERROR);
		RETURN;
	END_IF
	IF(THIS^.hasNext()) AND_THEN  THIS^.getNextTreeNode(node => THIS^.currentNode) THEN
		THIS^.currentObject := THIS^.currentNode.object;
		THIS^.processNode(THIS^.currentNode);
	ELSE
		cycleManager.proceedWith(SUCCESS);
		THIS^.currentObject := NULL;
	END_IF
END_CASE

iterate := cycleManager.state;
object := THIS^.currentObject;
END_METHOD

(*

## Short summary

This method is called when the node is taken from the nodelist.
Can perform actions as putting childnodes on the list etc.

.. <legal notes>

legal notes
=================
| SPDX-FileCopyrightText: © 2022 ekvip automation GmbH <info@ekvip.de>
| SPDX-License-Identifier: Apache-2.0
| For details check: Apache-2.0_

.. _Apache-2.0: https://www.apache.org/licenses/LICENSE-2.0

.. </legal notes>



*)

METHOD PROTECTED ABSTRACT processNode
VAR_INPUT
	nodeToProcess :CNM_CollectionInterfaces.IBinaryTreeNode;
END_VAR
END_METHOD

(*

## Short summary

This method is called in the initphase on the rootnode of the tree.
Default implementation executes processNode.

.. <legal notes>

legal notes
=================
| SPDX-FileCopyrightText: © 2025 ekvip automation GmbH <info@ekvip.de>
| SPDX-License-Identifier: Apache-2.0
| For details check: Apache-2.0_

.. _Apache-2.0: https://www.apache.org/licenses/LICENSE-2.0

.. </legal notes>



*)

METHOD PROTECTED processStartNode
VAR_INPUT
	nodeToProcess :CNM_CollectionInterfaces.IBinaryTreeNode;
END_VAR
THIS^.processNode(nodeToProcess);
END_METHOD

(*

## Short summary

This method resets the iterator. 
After a reset the iterator points to the first element if available.


**Example:**
```
iterator.reset();
WHILE(iterator.moveNext())DO
	foo := iterator.current.hashCode;
	bar := iterator.current.name;
END_WHILE
```

.. <legal notes>

legal notes
=================
| SPDX-FileCopyrightText: © 2022 ekvip automation GmbH <info@ekvip.de>
| SPDX-License-Identifier: Apache-2.0
| For details check: Apache-2.0_

.. _Apache-2.0: https://www.apache.org/licenses/LICENSE-2.0

.. </legal notes>

*)
METHOD reset
THIS^.iterate(FALSE);
THIS^.nodeList.clear();
THIS^.nodeList.append(THIS^.root);
THIS^.currentNode := THIS^.root;
THIS^.currentObject := 0;
END_METHOD

PROPERTY PROTECTED root : CNM_CollectionInterfaces.IBalancedBinarySearchTreeNode
GET
IF THIS^.isObjectValid(THIS^.tree) THEN
	root := THIS^.tree.rootNode;
ELSE
	root := 0;
END_IF
END_GET
END_PROPERTY

END_FUNCTION_BLOCK

// ---- Iterate/classes/AbstractIterator.TcPOU
(*

## Short summary

An abstract class to implement most basic iterator functions for use in custom Iterators.
Users still need to implement iterate and hasNext, as these depend on the data-stucture.
Iterate should take care to assign ``THIS^.current`` in their iterate implementation.

.. <legal notes>

legal notes
=================
| SPDX-FileCopyrightText: © 2024 ekvip automation GmbH <info@ekvip.de>
| SPDX-License-Identifier: Apache-2.0
| For details check: Apache-2.0_

.. _Apache-2.0: https://www.apache.org/licenses/LICENSE-2.0

.. </legal notes>



*)

FUNCTION_BLOCK ABSTRACT AbstractIterator EXTENDS CNM_AbstractObject.Object IMPLEMENTS CNM_CollectionInterfaces.IIterator
VAR
	{attribute 'no_copy'}
	currentObject :CNM_AbstractObject.IObject;
END_VAR

(*

## Short summary

This property returns the current element which the iterator points to.

**Attention:** 
	If current is used multiple times between two iterate calls, 
	current is only guarenteed to return an object that is actually in the list fo rthe first call to current that happens
	immediatly after the first iteration call.
	
**Example:**
```
WHILE(iterator.moveNext())DO
	foo := iterator.current.hashCode;
	bar := iterator.current.name;
END_WHILE
```

.. <legal notes>

legal notes
=================
| SPDX-FileCopyrightText: © 2022 ekvip automation GmbH <info@ekvip.de>
| SPDX-License-Identifier: Apache-2.0
| For details check: Apache-2.0_

.. _Apache-2.0: https://www.apache.org/licenses/LICENSE-2.0

.. </legal notes>

*)
PROPERTY current :CNM_AbstractObject.IObject
GET
current := THIS^.currentObject;
END_GET
SET // PROTECTED
THIS^.currentObject := current;
END_SET
END_PROPERTY

(*

## Short summary

This method returns the next object from the iterator and move the iterator to it.
If there is no next object, this should return NULL.

**Example:**
```
WHILE(iterator.hasNext())DO
	iterator.getNext().hashcode;
END_WHILE
```

.. <legal notes>

legal notes
=================
| SPDX-FileCopyrightText: © 2022 ekvip automation GmbH <info@ekvip.de>
| SPDX-License-Identifier: Apache-2.0
| For details check: Apache-2.0_

.. _Apache-2.0: https://www.apache.org/licenses/LICENSE-2.0

.. </legal notes>


**Return:** ``CNM_AbstractObject.IObject``: next object in collection, NULL if End of Collection is reached

*)

METHOD FINAL getNext :CNM_AbstractObject.IObject
THIS^.iterate(execute := TRUE );
getNext := THIS^.current;
END_METHOD

(*

## Short summary

This method returns if there exists another element to iterate to.

**Example:**
```
WHILE(iterator.hasNext())DO
	iterator.getNext().foo();
END_WHILE
```

.. <legal notes>

legal notes
=================
| SPDX-FileCopyrightText: © 2022 ekvip automation GmbH <info@ekvip.de>
| SPDX-License-Identifier: Apache-2.0
| For details check: Apache-2.0_

.. _Apache-2.0: https://www.apache.org/licenses/LICENSE-2.0

.. </legal notes>


**Return:** ``TRUE``: Iterator has a next object that can be fetched with getNext()
	``FALSE``: Iterator finished

*)

METHOD ABSTRACT hasNext :BOOL
END_METHOD

(*

## Short summary

This method delivers the next object from the collection and returns the current state of iteration.

**Example:**
You have a list: 1 2 3
the first iterate call will return CNM_ReturnTypes.BUSY and object = 1
the second iterate call will return CNM_ReturnTypes.BUSY and object = 2
the third iterate call will return CNM_ReturnTypes.BUSY and object = 3
the forth iterate call will return CNM_ReturnTypes.SUCCESS and object = NULL

**Attention:** iterators MUST assign the currently returned 'object' to ```THIS^.current``` as well! 

.. <legal notes>

legal notes
=================
| SPDX-FileCopyrightText: © 2022 ekvip automation GmbH <info@ekvip.de>
| SPDX-License-Identifier: Apache-2.0
| For details check: Apache-2.0_

.. _Apache-2.0: https://www.apache.org/licenses/LICENSE-2.0

.. </legal notes>


**Return:** ``SUCCESS``: if last object from collection was already returned,
    ``ABORTED``: execute has a falling edge during iterate,
    ``BUSY``: When iterate had rising edge on execute and not all objects had been returned yet,
    ``IDLE``: iterate wasn't started yet,
	``ERROR``: error occured during iteration
	
*)

METHOD ABSTRACT iterate :CNM_ReturnTypes.SingleExecutionState
VAR_INPUT
	(*control bit to start or abort the iterate (see SingleExecutionState)*)
	execute	:BOOL;
END_VAR
VAR_OUTPUT
	(*the returned object of the iteration*)
	object		:CNM_AbstractObject.IObject;
END_VAR
END_METHOD

(*

## Short summary

This method returns true if there exists another element to iterate to and fetches the next element to THIS^.current.
It return false if no further elements exist in the collection, in this case it sets THIS^.current to NULL.

**Example:**
```
WHILE(iterator.moveNext())DO
	iterator.current.foo();
END_WHILE
```

.. <legal notes>

legal notes
=================
| SPDX-FileCopyrightText: © 2022 ekvip automation GmbH <info@ekvip.de>
| SPDX-License-Identifier: Apache-2.0
| For details check: Apache-2.0_

.. _Apache-2.0: https://www.apache.org/licenses/LICENSE-2.0

.. </legal notes>


**Return:** ``TRUE``: Iterator had a next object that can be now accessed with current
	``FALSE``: Iterator finished, current will be NULL

*)

METHOD FINAL moveNext :BOOL
moveNext := THIS^.hasNext();
THIS^.getNext();
END_METHOD

(*

## Short summary

This method resets the iterator.

**Example:**
```
iterator.reset();
WHILE(iterator.moveNext())DO
	foo := iterator.current.hashCode;
	bar := iterator.current.name;
END_WHILE
```

.. <legal notes>

legal notes
=================
| SPDX-FileCopyrightText: © 2022 ekvip automation GmbH <info@ekvip.de>
| SPDX-License-Identifier: Apache-2.0
| For details check: Apache-2.0_

.. _Apache-2.0: https://www.apache.org/licenses/LICENSE-2.0

.. </legal notes>

*)

METHOD reset
THIS^.iterate(execute := FALSE);
END_METHOD

END_FUNCTION_BLOCK

// ---- Lists/LinkedList/classes/LinkedList.TcPOU
(*

## Short summary

Implementation of ILinkedList.
Does not allow empty objects as data!

**Warning:**
	Calling __DELETE directly on a Collection will bypass the destruct Context and therefore also delete the contained elements.

.. <legal notes>

legal notes
=================
| SPDX-FileCopyrightText: © 2022 ekvip automation GmbH <info@ekvip.de>
| SPDX-License-Identifier: Apache-2.0
| For details check: Apache-2.0_

.. _Apache-2.0: https://www.apache.org/licenses/LICENSE-2.0

.. </legal notes>



*)
{attribute 'enable_dynamic_creation'}
FUNCTION_BLOCK LinkedList EXTENDS AbstractList IMPLEMENTS ILinkedListHelpers
VAR
	headElement				:CNM_CollectionInterfaces.IDoublyLinkedElement;
	lastElement				:CNM_CollectionInterfaces.IDoublyLinkedElement;
	injectedSorter			:CNM_CollectionInterfaces.ILinkedListSorter;
	(*true if the sorter were created inside this list, false if set from outside*)
	listChangedDuringSort 	:BOOL	:= FALSE;
	listChangedIterate 		:BOOL	:= FALSE;
	
END_VAR

(*

## Short summary

This method is called every time the list changes and can notify other components.

.. <legal notes>

legal notes
=================
| SPDX-FileCopyrightText: © 2022 ekvip automation GmbH <info@ekvip.de>
| SPDX-License-Identifier: Apache-2.0
| For details check: Apache-2.0_

.. _Apache-2.0: https://www.apache.org/licenses/LICENSE-2.0

.. </legal notes>



*)

METHOD PROTECTED announceListChange
VAR_INPUT
END_VAR
THIS^.listChangedIterate := TRUE;
THIS^.changesToCollection := THIS^.changesToCollection+1;
END_METHOD

(*

## Short summary

This method adds the given object to the end of the list.
Adding NULL-Objects or THIS^ to the list is not possible.

.. <legal notes>

legal notes
=================
| SPDX-FileCopyrightText: © 2022 ekvip automation GmbH <info@ekvip.de>
| SPDX-License-Identifier: Apache-2.0
| For details check: Apache-2.0_

.. _Apache-2.0: https://www.apache.org/licenses/LICENSE-2.0

.. </legal notes>


**Return:** ``CNM_ReturnTypes.SingleExecutionResult.SUCCESS``: prepend was successful
	``CNM_ReturnTypes.SingleExecutionResult.ERROR``: allocation of container for new element failed, list not changed 
	``CNM_ReturnTypes.SingleExecutionResult.ABORTED``: NULL object or this list was passed

*)
METHOD append :CNM_ReturnTypes.SingleExecutionResult
VAR_INPUT
	(*The object to be appended*)
	object	:CNM_AbstractObject.IObject;
END_VAR
VAR
	newElement 	:CNM_CollectionInterfaces.IDoublyLinkedElement;
END_VAR
VAR CONSTANT
	IS_NOT_REFERENCED 	:__XWORD := 0;
END_VAR
append := CNM_ReturnTypes.SingleExecutionResult.ABORTED;
RETURN (THIS^.isObjectNull(object) OR THIS^.isEqual(object));
	
RETURN( 
	(append := THIS^.collectionFactory.getNewDoublyLinkedElement(
		object				:= object,
		previousElement		:= THIS^.lastElement,
		nextElement			:= IS_NOT_REFERENCED,
		linkElements		:= TRUE,
		element 			=> newElement)
	) <> CNM_ReturnTypes.SingleExecutionResult.SUCCESS 
);

THIS^.last := newElement;
IF(THIS^.isObjectNull(THIS^.head))THEN
	THIS^.head := THIS^.last;
END_IF

THIS^.incrementSize();
THIS^.announceListChange();
END_METHOD

(*

## Short summary

This method adds all elements of the given collection to the end of this list.

.. <legal notes>

legal notes
=================
| SPDX-FileCopyrightText: © 2025 ekvip automation GmbH <info@ekvip.de>
| SPDX-License-Identifier: Apache-2.0
| For details check: Apache-2.0_

.. _Apache-2.0: https://www.apache.org/licenses/LICENSE-2.0

.. </legal notes>


**Return:** ``CNM_ReturnTypes.SingleExecutionResult.SUCCESS``: new Container not needed / could be allocated and data was copied
	``CNM_ReturnTypes.SingleExecutionResult.ERROR``: new Container couldn't be allocated, container left unchanged
	``CNM_ReturnTypes.SingleExecutionResult.ABORTED``: NULL object or the list itself was passed

*)
METHOD appendCollection :CNM_ReturnTypes.SingleExecutionResult
VAR_INPUT
	(*The collection to be appended*)
	collectionToAppend	:CNM_CollectionInterfaces.ICollection;
END_VAR
VAR
	collectionElement 	:CNM_AbstractObject.IObject;
	oldLast				:CNM_CollectionInterfaces.IDoublyLinkedElement;
	destructElement		:CNM_CollectionInterfaces.IDoublyLinkedElement;
	nextElement			:CNM_CollectionInterfaces.IDoublyLinkedElement;
	iterator			:CNM_CollectionInterfaces.IIterator;
	iterateState		:CNM_ReturnTypes.SingleExecutionState;
END_VAR
VAR CONSTANT
	NULL :__XWORD := 0;
END_VAR
appendCollection := CNM_ReturnTypes.SingleExecutionResult.ABORTED;
RETURN(THIS^.isEqual(collectionToAppend) OR_ELSE THIS^.isObjectNull(collectionToAppend) );
oldLast := THIS^.last;
appendCollection := collectionToAppend.createNewIterator(iterator => iterator);
RETURN(appendCollection <> CNM_ReturnTypes.SingleExecutionResult.SUCCESS);
iterateState := iterator.iterate(FALSE);
iterateState := iterator.iterate(TRUE, object => collectionElement);
WHILE ((
		THIS^.isObjectValid(collectionElement)
	) AND (
		appendCollection = CNM_ReturnTypes.SingleExecutionResult.SUCCESS
	) AND (
		iterateState = CNM_ReturnTypes.SingleExecutionState.BUSY
	)
)DO
	appendCollection := THIS^.append(collectionElement);
	iteratestate := iterator.iterate(TRUE, object => collectionElement);
END_WHILE

IF (appendCollection = CNM_ReturnTypes.SingleExecutionResult.ERROR) THEN
	THIS^.last := oldLast;
	destructElement := oldLast.next;
	WHILE (THIS^.isObjectValid(destructElement)) DO
		nextElement := destructElement.next;
		destructElement.destruct();
		destructElement := nextElement;
	END_WHILE
	THIS^.last.next := NULL;
ELSE
	THIS^.announceListChange();
END_IF

IF THIS^.isObjectValid(iterator) THEN
	iterator.destruct();
END_IF
END_METHOD

(*

## Short summary

This abstract property returns the class name of the concrete object, 
which is useful to check the class name for ``__DELETE``.

.. <legal notes>

legal notes
=================
| SPDX-FileCopyrightText: © 2022 ekvip automation GmbH <info@ekvip.de>
| SPDX-License-Identifier: Apache-2.0
| For details check: Apache-2.0_

.. _Apache-2.0: https://www.apache.org/licenses/LICENSE-2.0

.. </legal notes>

*)
PROPERTY className : CNM_AbstractObject.ClassName
GET
className := 'CNM_Collections.LinkedList';
END_GET
END_PROPERTY

(*

## Short summary

This method clears all elements from this list. 

.. <legal notes>

legal notes
=================
| SPDX-FileCopyrightText: © 2022 ekvip automation GmbH <info@ekvip.de>
| SPDX-License-Identifier: Apache-2.0
| For details check: Apache-2.0_

.. _Apache-2.0: https://www.apache.org/licenses/LICENSE-2.0

.. </legal notes>



*)
METHOD clear
VAR
	currentElement	:CNM_CollectionInterfaces.IDoublyLinkedElement;
	elementToDelete	:CNM_CollectionInterfaces.IDoublyLinkedElement;
END_VAR
VAR CONSTANT
	IS_NOT_REFERENCED 	:__XWORD := 0;
END_VAR
currentElement := THIS^.head;
WHILE (THIS^.isObjectValid(currentElement)) DO
	elementToDelete := currentElement;
	currentElement := currentElement.next;
	elementToDelete.destruct();
END_WHILE

THIS^.head := IS_NOT_REFERENCED;
THIS^.last := IS_NOT_REFERENCED;
THIS^.collectionSize := 0;
THIS^.announceListChange();
END_METHOD

(*

## Short summary

This method is called in the destruct method and is intended to zero all references and interfaces that should not be destructed. 
To delete the collection with all its contents, use deepDestruct() instead of destruct().

.. <legal notes>

legal notes
=================
| SPDX-FileCopyrightText: © 2025 ekvip automation GmbH <info@ekvip.de>
| SPDX-License-Identifier: Apache-2.0
| For details check: Apache-2.0_

.. _Apache-2.0: https://www.apache.org/licenses/LICENSE-2.0

.. </legal notes>

*)
METHOD PROTECTED clearContents
VAR CONSTANT
	NULL	: __XWORD := 0;
END_VAR
THIS^.clear();
THIS^.injectedSorter := 0;
END_METHOD

(*

## Short summary

This method is used to create a new instance
of the object which has the same internal state as the object.
If the object is a container class, the references to the content objects
are not cloned for this there is the method `ICloneable.deepClone`.

If an object does not support cloning the return value is
``CNM_ReturnTypes.CloneResult.CLONE_IS_NOT_SUPPORTED``.

If there is not enough memory or the cloning fails because the
attribute enable dynamic creation was forgotten the return value is 
``CNM_ReturnTypes.CloneResult.FAILED``.

Only if the return value is ``CNM_ReturnTypes.CloneResult.SUCCESS``
the output ``clonedObject`` points to the new object
otherwise ``clonedObject`` is NULL.  

**Attention:** 
	For derivations: **If a derived class needs ``clone`` this method must be overwritten.**
	and don't forget the attribute ``{attribute 'enable_dynamic_creation'}``  

.. <legal notes>

legal notes
=================
| SPDX-FileCopyrightText: © 2022 ekvip automation GmbH <info@ekvip.de>
| SPDX-License-Identifier: Apache-2.0
| For details check: Apache-2.0_

.. _Apache-2.0: https://www.apache.org/licenses/LICENSE-2.0

.. </legal notes>


**Return:**``CNM_ReturnTypes.CloneResult.SUCCESS``: new object clone was created,
``CNM_ReturnTypes.CloneResult.FAILED``: object clone failed
``CNM_ReturnTypes.CloneResult.CLONE_IS_NOT_SUPPORTED``: object does not support cloning

*)
METHOD clone : CNM_AbstractObject.CNM_ReturnTypes.CloneResult
VAR_OUTPUT
	(* new object instance or NULL if somthing went wrong *)
	clonedObject		:CNM_AbstractObject.IObject;
END_VAR
VAR
	miniMe				:POINTER TO LinkedList;
	iterator			:CNM_CollectionInterfaces.IIterator;
	objectToAppend		:CNM_AbstractObject.IObject;
END_VAR
clone := CNM_ReturnTypes.CloneResult.FAILED;
miniMe := __NEW(LinkedList());
RETURN (miniMe = 0);
clone := CNM_ReturnTypes.CloneResult.SUCCESS;
clonedObject := miniMe^;
IF (THIS^.size > 0) THEN
	IF (THIS^.createNewIterator(iterator => iterator) = CNM_ReturnTypes.SingleExecutionResult.SUCCESS) THEN
		iterator.iterate(FALSE);
		WHILE (iterator.iterate(TRUE, object => objectToAppend) <> CNM_ReturnTypes.SingleExecutionState.SUCCESS) DO
			IF THIS^.isObjectValid(objectToAppend) THEN
				miniMe^.append(objectToAppend);
			ELSE
				iterator.destruct();
				clone := CNM_ReturnTypes.CloneResult.FAILED;
				miniMe^.deepDestruct();
				clonedObject := 0;
				RETURN;
			END_IF
		END_WHILE
		iterator.destruct();
	END_IF
END_IF
END_METHOD

(*

## Short summary

This method compares a foreign object with the own one, this is needed for sort orders.
The abstract class evaluates every object that is NULL as greater, and all other objects as equal. 

.. <legal notes>

legal notes
=================
| SPDX-FileCopyrightText: © 2022 ekvip automation GmbH <info@ekvip.de>
| SPDX-License-Identifier: Apache-2.0
| For details check: Apache-2.0_

.. _Apache-2.0: https://www.apache.org/licenses/LICENSE-2.0

.. </legal notes>


**Return:** ``SMALLER``: ``THIS`` precedes in order,
	``EQUAL``: ``THIS`` and ``object`` at the same position in order,
	``GREATER``: ``THIS`` is after in order.
	Checkout :``CNM_CollectionInterfaces.ComparationResult``.

*)
METHOD compareTo :CNM_ReturnTypes.ComparationResult
VAR_INPUT
	(*the object to be compared to*)
	object	:CNM_CollectionInterfaces.CNM_AbstractObject.IObject;
END_VAR
VAR
	collection :CNM_CollectionInterfaces.ICollection;
END_VAR
IF (THIS^.isObjectNull(object)) THEN
	compareTo := CNM_ReturnTypes.ComparationResult.GREATER;
ELSE
	compareTo := CNM_ReturnTypes.ComparationResult.EQUAL;
	IF(__QUERYINTERFACE(object, collection)) THEN
		IF(collection.size < THIS^.size) THEN
			compareTo := CNM_ReturnTypes.ComparationResult.GREATER;
		ELSIF(collection.size > THIS^.size) THEN
			compareTo := CNM_ReturnTypes.ComparationResult.SMALLER;			
		END_IF
	END_IF
END_IF
END_METHOD

(*

## Short summary

This method returns a NEW Iterator instance which can iterate the collection.
These iterators can be used parallel independend of each other on the same collection.

**Warning:**
The returned Iterator was created using the __NEW operator and must be destructed to avoid memory leaks!



.. <legal notes>

legal notes
=================
| SPDX-FileCopyrightText: © 2024 ekvip automation GmbH <info@ekvip.de>
| SPDX-License-Identifier: Apache-2.0
| For details check: Apache-2.0_

.. _Apache-2.0: https://www.apache.org/licenses/LICENSE-2.0

.. </legal notes>



*)
METHOD createNewIterator :CNM_CollectionInterfaces.CNM_ReturnTypes.SingleExecutionResult
VAR_OUTPUT
	(*The new created iterator or null if allocation fails *)
	iterator	:CNM_CollectionInterfaces.IIterator;
END_VAR
VAR
	newIterator :POINTER TO ForwardLinkedListIterator;
END_VAR
newIterator := __NEW(ForwardLinkedListIterator(list := THIS^));
IF (newIterator = 0) THEN
	createNewIterator := CNM_ReturnTypes.SingleExecutionResult.ERROR;
	RETURN;
END_IF
createNewIterator := CNM_ReturnTypes.SingleExecutionResult.SUCCESS;
iterator := newIterator^;
END_METHOD

(*

## Short summary

Reduces the collectionsize by one

.. <legal notes>

legal notes
=================
| SPDX-FileCopyrightText: © 2023 ekvip automation GmbH <info@ekvip.de>
| SPDX-License-Identifier: Apache-2.0
| For details check: Apache-2.0_

.. _Apache-2.0: https://www.apache.org/licenses/LICENSE-2.0

.. </legal notes>



*)

METHOD PROTECTED decrementSize
VAR_INPUT
END_VAR
THIS^.collectionSize := THIS^.collectionSize-1;
END_METHOD

(*

## Short summary

This method is used to create a new instance
of the object which has the same internal state as the object.
If the object is a container class, the references to the content objects
are cloned too.

If an object does not support cloning the return value is
``CNM_ReturnTypes.CloneResult.CLONE_IS_NOT_SUPPORTED``.

If there is not enough memory or the cloning fails because the
attribute enable dynamic creation was forgotten the return value is 
``CNM_ReturnTypes.CloneResult.FAILED``.
If something goes wrong, then this method must clean up everything
that has been cloned and free the memory again.
**The deepClone either works completely, or not at all**

Only if the return value is ``CNM_ReturnTypes.CloneResult.SUCCESS``
the output ``clonedObject`` points to the new object
otherwise ``clonedObject`` is NULL.  

**Attention:** 
	For derivations: **If a derived class needs ``deepClone`` this method must be overwritten.**
	and don't forget the attribute ``{attribute 'enable_dynamic_creation'}``, even for container content 

.. <legal notes>

legal notes
=================
| SPDX-FileCopyrightText: © 2022 ekvip automation GmbH <info@ekvip.de>
| SPDX-License-Identifier: Apache-2.0
| For details check: Apache-2.0_

.. _Apache-2.0: https://www.apache.org/licenses/LICENSE-2.0

.. </legal notes>


**Return:**``CNM_ReturnTypes.CloneResult.SUCCESS``: new object clone was created,
``CNM_ReturnTypes.CloneResult.FAILED``: object clone failed
``CNM_ReturnTypes.CloneResult.CLONE_IS_NOT_SUPPORTED``: object does not support deep cloning

*)
METHOD deepClone : CNM_AbstractObject.CNM_ReturnTypes.CloneResult
VAR_OUTPUT
	(* new object instance or NULL if somthing went wrong *)
	clonedObject		:CNM_AbstractObject.IObject;
END_VAR
VAR
	miniMe				:POINTER TO LinkedList;
	iterator			:CNM_CollectionInterfaces.IIterator;
	objectToClone		:CNM_AbstractObject.IObject;
	clonedObj			:CNM_AbstractObject.IObject;
	clonedSorterObject	:CNM_AbstractObject.IObject;
	clonedSorter		:CNM_CollectionInterfaces.ILinkedListSorter;
	tmpResult 			:CNM_ReturnTypes.CloneResult;
	allObjectsValid		:BOOL	:= TRUE;
END_VAR
deepClone := CNM_ReturnTypes.CloneResult.FAILED;
miniMe := __NEW(LinkedList());
RETURN (miniMe = 0);
deepClone := CNM_ReturnTypes.CloneResult.SUCCESS;
clonedObject := miniMe^;
IF (THIS^.size > 0) THEN
	IF (THIS^.createNewIterator(iterator => iterator) = CNM_ReturnTypes.SingleExecutionResult.SUCCESS) THEN
		iterator.iterate(FALSE);
		WHILE (iterator.iterate(TRUE, object => objectToClone) = CNM_ReturnTypes.SingleExecutionState.BUSY) DO
			allObjectsValid := allObjectsValid AND THIS^.isObjectValid(objectToClone);
		END_WHILE
		IF allObjectsValid THEN
			iterator.iterate(FALSE);
			WHILE (iterator.iterate(TRUE, object => objectToClone) <> CNM_ReturnTypes.SingleExecutionState.SUCCESS) DO
				IF THIS^.isObjectValid(objectToClone) THEN
					tmpResult := objectToClone.deepClone(clonedObject => clonedObj); 
					IF ( tmpResult = CNM_ReturnTypes.CloneResult.SUCCESS) THEN
						miniMe^.append(clonedObj);
					ELSE
						iterator.destruct();
						deepClone := tmpResult;
						miniMe^.deepDestruct();
						clonedObject := 0;
						RETURN;
					END_IF
				END_IF
			END_WHILE
		ELSE
			deepClone := CNM_ReturnTypes.CloneResult.FAILED;
			miniMe^.deepDestruct();
			clonedObject := 0;
			RETURN;
		END_IF
		iterator.destruct();
	END_IF
END_IF

RETURN (THIS^.isObjectNull(THIS^.injectedSorter));
tmpResult := THIS^.injectedSorter.deepClone(clonedObject => clonedSorterObject);
IF ((tmpResult <> CNM_ReturnTypes.CloneResult.SUCCESS) 
		OR_ELSE 
	THIS^.isObjectNull(clonedSorterObject) 
		OR_ELSE 
	(NOT __QUERYINTERFACE(clonedSorterObject, clonedSorter))
) THEN
	deepClone := SEL((tmpResult = CNM_ReturnTypes.CloneResult.SUCCESS), tmpResult, CNM_ReturnTypes.CloneResult.FAILED);
	miniMe^.deepDestruct();
	clonedObject := 0;
	RETURN;
END_IF

miniMe^.setSorter(sorter := clonedSorter);
deepClone := CNM_ReturnTypes.CloneResult.SUCCESS;
END_METHOD

(*

## Short summary

This property returns the last object in the first and removes it from the list. Can be seen as opposite of prepend.
**Example:**
On a list: (Head -->) A B C, list.dequeue will return A.
**Example 2:**
If you call prepend(x), a dequeue right after will return x.

.. <legal notes>

legal notes
=================
| SPDX-FileCopyrightText: © 2022 ekvip automation GmbH <info@ekvip.de>
| SPDX-License-Identifier: Apache-2.0
| For details check: Apache-2.0_

.. _Apache-2.0: https://www.apache.org/licenses/LICENSE-2.0

.. </legal notes>

*)

METHOD dequeue :CNM_AbstractObject.IObject
VAR_INPUT
END_VAR
VAR
	oldHead		:CNM_CollectionInterfaces.IDoublyLinkedElement;
END_VAR
VAR CONSTANT
	IS_NOT_REFERENCED 	:__XWORD := 0;
END_VAR
dequeue := IS_NOT_REFERENCED;
IF (THIS^.isObjectValid(THIS^.head)) THEN
	dequeue		:= THIS^.head.object;
	oldHead		:= THIS^.head;
	THIS^.head	:= oldHead.next;	
	oldHead.destruct();
	IF (THIS^.isObjectNull(THIS^.head)) THEN
		THIS^.last := IS_NOT_REFERENCED;
	END_IF;
	THIS^.decrementSize();
	THIS^.announceListChange();
END_IF
END_METHOD

(*

## Short summary

Destructs the passed element. Next and Previous Element are relinked to prevent gaps. Also takes care that head / last are updated if necessary

.. <legal notes>

legal notes
=================
| SPDX-FileCopyrightText: © 2023 ekvip automation GmbH <info@ekvip.de>
| SPDX-License-Identifier: Apache-2.0
| For details check: Apache-2.0_

.. _Apache-2.0: https://www.apache.org/licenses/LICENSE-2.0

.. </legal notes>



*)

METHOD PROTECTED destructLinkedElement
VAR_INPUT
	(*The element that should be destructed*)
	element :CNM_CollectionInterfaces.IDoublyLinkedElement;
END_VAR
IF(THIS^.isObjectNull(element))THEN
	RETURN;
END_IF
IF (THIS^.isObjectValid(THIS^.head) AND_THEN THIS^.head.isEqual(element)) THEN
	THIS^.head := THIS^.head.next;
END_IF
IF (THIS^.isObjectValid(THIS^.lastElement) AND_THEN THIS^.last.isEqual(element)) THEN
	THIS^.lastElement := THIS^.lastElement.previous;
END_IF
IF (THIS^.isObjectValid(element.previous)) THEN
	element.previous.next := element.next;
END_IF
IF THIS^.isObjectValid(element.next) THEN
	 element.next.previous := element.previous;
END_IF
element.destruct();
END_METHOD

(*

## Short summary

Mark the object as deleted, as it staiys in the memory.

.. <legal notes>

legal notes
=================
| SPDX-FileCopyrightText: © 2022 ekvip automation GmbH <info@ekvip.de>
| SPDX-License-Identifier: Apache-2.0
| For details check: Apache-2.0_

.. _Apache-2.0: https://www.apache.org/licenses/LICENSE-2.0

.. </legal notes>

*)
METHOD FB_Exit : BOOL
VAR_INPUT
	(* TRUE: the exit method is called in order to leave the instance which will be copied afterwards (online change).*)
	bInCopyCode	: BOOL;
END_VAR
VAR
	currentElement 	:CNM_CollectionInterfaces.IDoublyLinkedElement;
	next 			:CNM_CollectionInterfaces.IDoublyLinkedElement;
END_VAR
currentElement := THIS^.head;
WHILE (THIS^.isObjectValid(currentElement)) DO
	next := currentElement.next;
	currentElement.deepDestruct();
	currentElement := next;
END_WHILE
IF THIS^.isObjectValid(THIS^.injectedSorter) THEN
	THIS^.injectedSorter.deepDestruct();
END_IF
END_METHOD

(*

## Short summary

Searches the containerobject, that contains a specific Element that is passed to the method.

.. <legal notes>

legal notes
=================
| SPDX-FileCopyrightText: © 2023 ekvip automation GmbH <info@ekvip.de>
| SPDX-License-Identifier: Apache-2.0
| For details check: Apache-2.0_

.. _Apache-2.0: https://www.apache.org/licenses/LICENSE-2.0

.. </legal notes>


**Return:** The (first) IDoublyLinkedElement that contains the ``object``, NULL if ``object`` is not contained in the list

*)

METHOD PROTECTED findObject :CNM_CollectionInterfaces.IDoublyLinkedElement
VAR_INPUT
	(*The object to search for*)
	object :CNM_AbstractObject.IObject;
END_VAR
VAR
	element	:CNM_CollectionInterfaces.IDoublyLinkedElement;
END_VAR
VAR CONSTANT
	IS_NOT_REFERENCED 	:__XWORD := 0;
END_VAR
IF(THIS^.isObjectNull(object))THEN
	findObject := IS_NOT_REFERENCED;
	RETURN;
END_IF
element := THIS^.head;
WHILE (THIS^.isObjectValid(element) AND_THEN NOT element.object.isEqual(object)) DO
	element := element.next;
END_WHILE
findObject := element;
END_METHOD

PROPERTY INTERNAL head : CNM_CollectionInterfaces.IDoublyLinkedElement
GET
head := THIS^.headElement;
END_GET
SET
THIS^.headElement := head;
END_SET
END_PROPERTY

(*

## Short summary

Increments the size of the list

.. <legal notes>

legal notes
=================
| SPDX-FileCopyrightText: © 2023 ekvip automation GmbH <info@ekvip.de>
| SPDX-License-Identifier: Apache-2.0
| For details check: Apache-2.0_

.. _Apache-2.0: https://www.apache.org/licenses/LICENSE-2.0

.. </legal notes>



*)
METHOD PROTECTED incrementSize
VAR_INPUT
END_VAR
THIS^.collectionSize := THIS^.collectionSize+1;
END_METHOD

METHOD INTERNAL instantSorting : CNM_ReturnTypes.SingleExecutionResult
VAR_INPUT
	order :SortingOrder;
	(*Optional: the comparator that should be used for the sort. Must not be changed while sort is in process*)
	comparator	: CNM_CollectionInterfaces.CNM_AbstractObject.IComparator := 0;
END_VAR
CASE order OF
SortingOrder.ASCENDING:
	instantSorting := THIS^.sorter.instantSort(
		size := THIS^.size,
		comparator := comparator,
		head := THIS^.headElement,
		last := THIS^.lastElement,
		currentListVersion := THIS^.changesToCollection
	);
SortingOrder.DESCENDING:
	instantSorting := THIS^.sorter.instantInverseSort(
		size := THIS^.size,
		comparator := comparator,
		head := THIS^.headElement,
		last := THIS^.lastElement,
		currentListVersion := THIS^.changesToCollection
	);
END_CASE
END_METHOD


(*

## Short summary

Inverts the List, so last element becomes first.
So List A B C D will be
D C B A

.. <legal notes>

legal notes
=================
| SPDX-FileCopyrightText: © 2022 ekvip automation GmbH <info@ekvip.de>
| SPDX-License-Identifier: Apache-2.0
| For details check: Apache-2.0_

.. _Apache-2.0: https://www.apache.org/licenses/LICENSE-2.0

.. </legal notes>



*)

METHOD invert
VAR
	leftElement 	:CNM_CollectionInterfaces.IDoublyLinkedElement;
	rightElement	:CNM_CollectionInterfaces.IDoublyLinkedElement;
	tmpElement 		:CNM_AbstractObject.IObject;
	index 			:UDINT;
	middle 			:UDINT;
END_VAR
RETURN(THIS^.size < 2);
leftElement := THIS^.head;
rightElement := THIS^.last;

middle := SHR(THIS^.size,1);
FOR index := 1 TO middle DO
	tmpElement := leftElement.object;
	leftElement.object := rightElement.object;
	rightElement.object := tmpElement;
	leftElement := leftElement.next;
	rightElement := rightElement.previous;
END_FOR

THIS^.announceListChange();
END_METHOD

(*

## Short summary

This method returns the next object in the iteration and returns an execution state.

.. <legal notes>

legal notes
=================
| SPDX-FileCopyrightText: © 2022 ekvip automation GmbH <info@ekvip.de>
| SPDX-License-Identifier: Apache-2.0
| For details check: Apache-2.0_

.. _Apache-2.0: https://www.apache.org/licenses/LICENSE-2.0

.. </legal notes>


**Return:** ``SUCCESS``: if last object from collection was returned,
	``ABORTED``: execute has a falling edge during iterate,
	``BUSY``: When iterate had rising edge on execute and not all objects had been returned yet
	``IDLE``: iterate not in progress, execute is false and iterate reseted 

*)
METHOD PROTECTED iterate :CNM_ReturnTypes.SingleExecutionState
VAR_INPUT
	(*False to init, True to retrieve next element*)
	execute	: BOOL;
END_VAR
VAR_OUTPUT
	(*The current element of the iteration*)
	object	:CNM_AbstractObject.IObject;
END_VAR
VAR_INST
	currentElement		:CNM_CollectionInterfaces.IDoublyLinkedElement;
	cycleManager		:CNM_CycleManager.SimpleCycleManager;
	currentListVersion 	:__XWORD;
END_VAR
VAR CONSTANT
	IS_NOT_REFERENCED 	:__XWORD := 0;
	INIT 		:DINT := CNM_ReturnTypes.DefaultSteps.STEP.INIT;
	ITERATING 	:DINT := INIT +1;
	ERROR		:DINT := CNM_ReturnTypes.DefaultSteps.STEP.ERROR;
END_VAR
IF (cycleManager.step.current > INIT) THEN
	cycleManager.assert.bitNumber.x.valueIsEqualTo(
		currentValue := currentListVersion,
		expectedValue := THIS^.changesToCollection,
		message := 'This instance of LinkedList has changed between iterate calls'
	);
END_IF

cycleManager(execute := execute);
CASE cycleManager.step.current OF
INIT:
	currentElement := THIS^.head;	
	currentListVersion := THIS^.changesToCollection;
	IF (THIS^.isObjectValid(currentElement)) THEN
		object := currentElement.object;
		currentElement := currentElement.next;
		cycleManager.proceed();
	ELSE
		cycleManager.proceedWith(CNM_ReturnTypes.DefaultSteps.STEP.SUCCESS);
	END_IF			
ITERATING:
	IF (THIS^.isObjectValid(currentElement)) THEN
		object := currentElement.object;
		currentElement := currentElement.next;
	ELSE
		cycleManager.proceedWith(CNM_ReturnTypes.DefaultSteps.STEP.SUCCESS);
	END_IF
ERROR:
	object := IS_NOT_REFERENCED; 
END_CASE

iterate := cycleManager.state;
END_METHOD

PROPERTY INTERNAL last : CNM_CollectionInterfaces.IDoublyLinkedElement
GET
last := THIS^.lastElement;
END_GET
SET
THIS^.lastElement := last;
END_SET
END_PROPERTY

(*

## Short summary

Links the passed element together with the other two passed element
Does not only adds the links to element, but also sets next.previous to element and previous.next to element,
to ensure a consistent list

.. <legal notes>

legal notes
=================
| SPDX-FileCopyrightText: © 2023 ekvip automation GmbH <info@ekvip.de>
| SPDX-License-Identifier: Apache-2.0
| For details check: Apache-2.0_

.. _Apache-2.0: https://www.apache.org/licenses/LICENSE-2.0

.. </legal notes>



*)
METHOD PROTECTED linkElement
VAR_INPUT
	(*the element that should be set as previous element*)
	previous		:CNM_CollectionInterfaces.IDoublyLinkedElement	:= IS_NOT_REFERENCED;
	(*The element that should be new linked*)
	element		:CNM_CollectionInterfaces.IDoublyLinkedElement	:= IS_NOT_REFERENCED;
	(*The element that should be used as next element*)
	next			:CNM_CollectionInterfaces.IDoublyLinkedElement	:= IS_NOT_REFERENCED;	
END_VAR
VAR CONSTANT
	IS_NOT_REFERENCED	:__UXINT := 0;
END_VAR
IF (THIS^.isObjectNull(element)) THEN
	RETURN;
END_IF

element.previous	:= previous;
element.next			:= next;

IF (THIS^.isObjectValid(previous)) THEN
	previous.next := element;
END_IF
IF (THIS^.isObjectValid(next)) THEN
	next.previous := element;
END_IF
END_METHOD

PROPERTY INTERNAL listChangeIndex : __XWORD
GET
listChangeIndex := THIS^.changesToCollection;
END_GET
SET
THIS^.changesToCollection := listChangeIndex;
END_SET
END_PROPERTY

(*

## Short summary

This property returns the last object in the list and removes it from the list. Can be seen as opposite of append.
**Example:**
On a list: (Head -->) A B C, list.pop will return C.
**Example 2:**
If you call append(x), a pop right after will return x.

.. <legal notes>

legal notes
=================
| SPDX-FileCopyrightText: © 2022 ekvip automation GmbH <info@ekvip.de>
| SPDX-License-Identifier: Apache-2.0
| For details check: Apache-2.0_

.. _Apache-2.0: https://www.apache.org/licenses/LICENSE-2.0

.. </legal notes>

*)

METHOD pop :CNM_AbstractObject.IObject
VAR_INPUT
END_VAR
VAR
	oldLast		:CNM_CollectionInterfaces.IDoublyLinkedElement;
END_VAR
VAR CONSTANT
	IS_NOT_REFERENCED 	:__XWORD := 0;
END_VAR
pop := IS_NOT_REFERENCED;

IF (THIS^.isObjectValid(THIS^.last)) THEN
	pop 		:= THIS^.last.object;
	oldLast		:= THIS^.lastElement;
	THIS^.last	:= THIS^.last.previous;
	oldLast.destruct();
	IF (THIS^.isObjectNull(THIS^.last)) THEN
		THIS^.head := IS_NOT_REFERENCED;
	ELSE
		THIS^.last.next := IS_NOT_REFERENCED;
	END_IF;	
	THIS^.decrementSize();
	THIS^.announceListChange();
END_IF
END_METHOD

(*

## Short summary

This method adds the given object as new head to the list.
Adding NULL-Objects or THIS^ to the list is not possible. 

.. <legal notes>

legal notes
=================
| SPDX-FileCopyrightText: © 2022 ekvip automation GmbH <info@ekvip.de>
| SPDX-License-Identifier: Apache-2.0
| For details check: Apache-2.0_

.. _Apache-2.0: https://www.apache.org/licenses/LICENSE-2.0

.. </legal notes>


**Return:** ``CNM_ReturnTypes.SingleExecutionResult.SUCCESS``: new Container not needed / could be allocated and data was copied
	``CNM_ReturnTypes.SingleExecutionResult.ERROR``: new Container couldn't be allocated, container left unchanged
	``CNM_ReturnTypes.SingleExecutionResult.ABORTED``: NULL object or the list itself was passed
*)
METHOD prepend :CNM_ReturnTypes.SingleExecutionResult
VAR_INPUT
	(*The object to be prepended*)
	object	: CNM_CollectionInterfaces.CNM_AbstractObject.IObject;
END_VAR
VAR
	result :CNM_ReturnTypes.SingleExecutionResult;
	newElement 	:CNM_CollectionInterfaces.IDoublyLinkedElement;
END_VAR
VAR CONSTANT
	IS_NOT_REFERENCED : __XWORD := 0;
END_VAR
prepend := CNM_ReturnTypes.SingleExecutionResult.ABORTED;
RETURN (THIS^.isObjectNull(object) OR THIS^.isEqual(object));	
RETURN( 
	(prepend := THIS^.collectionFactory.getNewDoublyLinkedElement(
		object				:= object,
		previousElement		:= IS_NOT_REFERENCED,
		nextElement			:= THIS^.headElement,
		linkElements		:= TRUE,
		element 			=> newElement)
	) <> CNM_ReturnTypes.SingleExecutionResult.SUCCESS 
);
THIS^.head := newElement;
IF(THIS^.isObjectNull(THIS^.last))THEN
	THIS^.last := THIS^.head;
END_IF
THIS^.incrementSize();
THIS^.announceListChange();
END_METHOD

(*

## Short summary

This method adds all elements of the given collection to the start of this list. 

.. <legal notes>

legal notes
=================
| SPDX-FileCopyrightText: © 2025 ekvip automation GmbH <info@ekvip.de>
| SPDX-License-Identifier: Apache-2.0
| For details check: Apache-2.0_

.. _Apache-2.0: https://www.apache.org/licenses/LICENSE-2.0

.. </legal notes>


**Return:** ``CNM_ReturnTypes.SingleExecutionResult.SUCCESS``: prepend was successful
	``CNM_ReturnTypes.SingleExecutionResult.ERROR``: collection to prepend didn't fit in old container, and new container couldn't be allocated
	``CNM_ReturnTypes.SingleExecutionResult.ABORTED``: NULL object or this arraylist was passed
	

*)
METHOD prependCollection :CNM_ReturnTypes.SingleExecutionResult
VAR_INPUT
	(*The collection to be prepended*)
	collectionToPrepend		:CNM_CollectionInterfaces.ICollection;
END_VAR
VAR
	collectionElement 		:CNM_AbstractObject.IObject;
	oldHead 				:CNM_CollectionInterfaces.IDoublyLinkedElement;
	current 				:CNM_CollectionInterfaces.IDoublyLinkedElement;
	old 					:CNM_CollectionInterfaces.IDoublyLinkedElement;
	newElement 				:CNM_CollectionInterfaces.IDoublyLinkedElement;
	iterator				:CNM_CollectionInterfaces.IIterator;
	result					:CNM_ReturnTypes.SingleExecutionResult;
	iterateState			:CNM_ReturnTypes.SingleExecutionState;
END_VAR
VAR CONSTANT
	IS_NOT_REFERENCED 		:__XWORD := 0;
END_VAR
prependCollection := CNM_ReturnTypes.SingleExecutionResult.ABORTED;
RETURN(THIS^.isObjectNull(collectionToPrepend) OR_ELSE THIS^.isEqual(collectionToPrepend));

RETURN((prependCollection := collectionToPrepend.createNewIterator(iterator => iterator)) <> CNM_ReturnTypes.SingleExecutionResult.SUCCESS);

iterateState := iterator.iterate(FALSE);

oldHead := THIS^.headElement;
iterateState := iterator.iterate(TRUE, object => collectionElement);
result := THIS^.collectionFactory.getNewDoublyLinkedElement(
	object				:= collectionElement,
	previousElement		:= IS_NOT_REFERENCED,
	nextElement			:= IS_NOT_REFERENCED,
	linkElements		:= TRUE,
	element				=> newElement
);

THIS^.head := newElement;
current := newElement;
IF THIS^.isObjectNull(current) THEN
	prependCollection := CNM_ReturnTypes.SingleExecutionResult.ERROR;
END_IF

iterateState := iterator.iterate(TRUE, object => collectionElement);
WHILE((
		THIS^.isObjectValid(collectionElement) 
	) AND ( 
		prependCollection = CNM_ReturnTypes.SingleExecutionResult.SUCCESS
	) AND (
		iterateState = CNM_ReturnTypes.SingleExecutionState.BUSY
	)
)DO
	result := THIS^.collectionFactory.getNewDoublyLinkedElement(
		object				:= collectionElement,
		previousElement		:= current,
		nextElement			:= IS_NOT_REFERENCED,
		linkElements		:= TRUE,
		element				=> newElement				
	);
	current := newElement;
	iterateState := iterator.iterate(TRUE, object => collectionElement);
END_WHILE

//in case of failed reset to old state
IF (prependCollection = CNM_ReturnTypes.SingleExecutionResult.ERROR) THEN
	WHILE THIS^.isObjectValid(current) DO
		old := current;
		current := current.previous;
		old.destruct();
	END_WHILE
	THIS^.head := oldHead;
	RETURN; 
END_IF

current.next := oldHead;
IF(THIS^.isObjectValid(oldHead))THEN
	oldHead.previous := current;	
ELSE
	THIS^.last := current;
END_IF

THIS^.collectionSize := (THIS^.collectionSize + collectionToPrepend.size);
THIS^.announceListChange();
IF THIS^.isObjectValid(iterator) THEN
	iterator.destruct();
END_IF
END_METHOD

(*

## Short summary

This method removes the first occurrence of the given object from the list.

.. <legal notes>

legal notes
=================
| SPDX-FileCopyrightText: © 2022 ekvip automation GmbH <info@ekvip.de>
| SPDX-License-Identifier: Apache-2.0
| For details check: Apache-2.0_

.. _Apache-2.0: https://www.apache.org/licenses/LICENSE-2.0

.. </legal notes>



*)
METHOD remove
VAR_INPUT
	(*The object to be removed from the list*)
	object	: CNM_CollectionInterfaces.CNM_AbstractObject.IObject;
END_VAR
VAR
	element	:CNM_CollectionInterfaces.IDoublyLinkedElement;
END_VAR
element := THIS^.findObject(object);
RETURN(THIS^.isObjectNull(element));
THIS^.destructLinkedElement(element);
THIS^.decrementSize();
THIS^.announceListChange();
END_METHOD

(*

## Short summary

This method can replace the default sorter for a custom one. Check ``IListSorter``
	
.. warning
	If the injected sorter was created dynamically,
	it will be automatically destruced within the deepdestruct context of THIS list.
	
.. <legal notes>

legal notes
=================
| SPDX-FileCopyrightText: © 2022 ekvip automation GmbH <info@ekvip.de>
| SPDX-License-Identifier: Apache-2.0
| For details check: Apache-2.0_

.. _Apache-2.0: https://www.apache.org/licenses/LICENSE-2.0

.. </legal notes>


**Return:** ``THIS`` :``ISortable``

*)
METHOD setSorter : CNM_CollectionInterfaces.ISortable
VAR_INPUT
	(*The instance of the sorter to be used to sort the list*)
	sorter	: CNM_CollectionInterfaces.ILinkedListSorter;
END_VAR
THIS^.injectedSorter := sorter;
setSorter := THIS^.sort;
END_METHOD

PROPERTY PROTECTED sorter :CNM_CollectionInterfaces.ILinkedListSorter
GET
VAR_INST
	instSorter :LinkedListMergeSorter;
END_VAR
IF(THIS^.isObjectValid(THIS^.injectedSorter))THEN
	sorter := THIS^.injectedSorter;
ELSE
	sorter := instSorter;
END_IF
END_GET
END_PROPERTY

METHOD INTERNAL sorting : CNM_ReturnTypes.SingleExecutionState
VAR_INPUT
	execute :BOOL;
	order :SortingOrder;
	(*Optional: the comparator that should be used for the sort. Must not be changed while sort is in process*)
	comparator	: CNM_CollectionInterfaces.CNM_AbstractObject.IComparator := 0;
END_VAR
CASE order OF
SortingOrder.ASCENDING:
	sorting := THIS^.sorter.sort(
		execute := execute,
		size := THIS^.size,
		comparator := comparator,
		head := THIS^.headElement,
		last := THIS^.lastElement,
		currentListVersion := THIS^.changesToCollection
	);
	
SortingOrder.DESCENDING:
	sorting := THIS^.sorter.inverseSort(
		execute := execute,
		size := THIS^.size,
		comparator := comparator,
		head := THIS^.headElement,
		last := THIS^.lastElement,
		currentListVersion := THIS^.changesToCollection
	);
END_CASE
END_METHOD

END_FUNCTION_BLOCK

// ---- Lists/LinkedList/classes/LinkedListIterator/classes/ForwardLinkedListIterator.TcPOU
{attribute 'enable_dynamic_creation'}
FUNCTION_BLOCK ForwardLinkedListIterator EXTENDS AbstractLinkedListIterator
VAR	
	lastChangeVersion :__XWORD;
	lastExecute :BOOL;
END_VAR

PROPERTY className :CNM_AbstractObject.ClassName
GET
className := 'ForwardLinkedListIterator';
END_GET
END_PROPERTY

(*

## Short summary

The constructor ``FB_init`` is needed to create an unique hash code.
The hash code is a pseudo random number create with a [xorshift](https://en.wikipedia.org/wiki/Xorshift) algorithm.
It can be overwritten on derivations, because it will be called implicit, ``SUPER^.FB_init()`` is not required.
For more information check: [Behavoir with derived function blocks](https://infosys.beckhoff.com/content/1033/tc3_plc_intro/5482088715.html?id=6983869892358031022).

.. <legal notes>

legal notes
=================
| SPDX-FileCopyrightText: © 2022 ekvip automation GmbH <info@ekvip.de>
| SPDX-License-Identifier: Apache-2.0
| For details check: Apache-2.0_

.. _Apache-2.0: https://www.apache.org/licenses/LICENSE-2.0

.. </legal notes>



*)
METHOD FB_init : BOOL
VAR_INPUT
	(* if TRUE, the retain variables are initialized (warm start / cold start)*)
	bInitRetains	: BOOL;
	(* if TRUE, the instance afterwards gets moved into the copy code (online change) *)
	bInCopyCode	: BOOL;
	(* list that is used to iterate*)
	list :REFERENCE TO LinkedList;
END_VAR
THIS^.direction := IterationDirection.FORWARD;
END_METHOD

END_FUNCTION_BLOCK

// ---- Lists/LinkedList/classes/LinkedListIterator/classes/AbstractLinkedListIterator.TcPOU
FUNCTION_BLOCK ABSTRACT AbstractLinkedListIterator EXTENDS AbstractIterator IMPLEMENTS ILinkedListIterator
VAR	
	{attribute 'hide'}
	list 				:REFERENCE TO LinkedList;
	currentElement		:CNM_CollectionInterfaces.IDoublyLinkedElement;
	direction 			:IterationDirection;
END_VAR

METHOD attachLinkedList : CNM_ReturnTypes.SingleExecutionResult
VAR_INPUT
	list :REFERENCE TO LinkedList;	
END_VAR
VAR CONSTANT
	NULL :CNM_AbstractObject.IObject := 0;
END_VAR
THIS^.currentElement := 0;
THIS^.current := 0;
attachLinkedList := CNM_ReturnTypes.SingleExecutionResult.ABORTED;
IF THIS^.isObjectValid(list) THEN
	THIS^.list REF= list;
	THIS^.currentElement := SEL(THIS^.direction = IterationDirection.BACKWARD, list.head, list.last);
	THIS^.currentObject := SEL(THIS^.isObjectValid(THIS^.currentElement), NULL, THIS^.currentElement.object);
	attachLinkedList := CNM_ReturnTypes.SingleExecutionResult.SUCCESS;
END_IF
END_METHOD

(*

## Short summary

The constructor ``FB_init`` is needed to create an unique hash code.
The hash code is a pseudo random number create with a [xorshift](https://en.wikipedia.org/wiki/Xorshift) algorithm.
It can be overwritten on derivations, because it will be called implicit, ``SUPER^.FB_init()`` is not required.
For more information check: [Behavoir with derived function blocks](https://infosys.beckhoff.com/content/1033/tc3_plc_intro/5482088715.html?id=6983869892358031022).

.. <legal notes>

legal notes
=================
| SPDX-FileCopyrightText: © 2022 ekvip automation GmbH <info@ekvip.de>
| SPDX-License-Identifier: Apache-2.0
| For details check: Apache-2.0_

.. _Apache-2.0: https://www.apache.org/licenses/LICENSE-2.0

.. </legal notes>



*)
METHOD FB_init : BOOL
VAR_INPUT
	(* if TRUE, the retain variables are initialized (warm start / cold start)*)
	bInitRetains	: BOOL;
	(* if TRUE, the instance afterwards gets moved into the copy code (online change) *)
	bInCopyCode	: BOOL;
	(* list that is used to iterate*)
	list :REFERENCE TO LinkedList;
END_VAR
VAR CONSTANT
	NULL :__XWORD := 0;
END_VAR
THIS^.list REF= list;
THIS^.currentObject := NULL;
IF THIS^.isObjectValid(THIS^.list) THEN
	THIS^.currentElement := SEL(THIS^.direction = IterationDirection.BACKWARD, THIS^.list.head, THIS^.list.last);
END_IF
END_METHOD

(*

## Short summary

This method returns if there exists another element to iterate to.

**Example:**
```
WHILE(iterator.hasNext())DO
	iterator.getNext().foo();
END_WHILE
```

.. <legal notes>

legal notes
=================
| SPDX-FileCopyrightText: © 2022 ekvip automation GmbH <info@ekvip.de>
| SPDX-License-Identifier: Apache-2.0
| For details check: Apache-2.0_

.. _Apache-2.0: https://www.apache.org/licenses/LICENSE-2.0

.. </legal notes>


**Return:** ``TRUE``: Iterator has a next object that can be fetched with getNext()
	``FALSE``: Iterator finished

*)
METHOD hasNext : BOOL
hasNext := 
THIS^.isObjectValid(THIS^.currentElement) 
	AND_THEN 
THIS^.isObjectValid(THIS^.currentElement.object);
END_METHOD

(*

## Short summary

This method returns the next object in the iteration and returns an execution state.
**Example:**
You have a list: 1 2 3
the first iterate call will return CNM_ReturnTypes.BUSY and object = 1
the second iterate call will return CNM_ReturnTypes.BUSY and object = 2
the third iterate call will return CNM_ReturnTypes.BUSY and object = 3
the forth iterate call will return CNM_ReturnTypes.SUCCESS and object = NULL

.. <legal notes>

legal notes
=================
| SPDX-FileCopyrightText: © 2022 ekvip automation GmbH <info@ekvip.de>
| SPDX-License-Identifier: Apache-2.0
| For details check: Apache-2.0_

.. _Apache-2.0: https://www.apache.org/licenses/LICENSE-2.0

.. </legal notes>


**Return:** ``SingleExecutionState.SUCCESS``: Iteration finished, no new elements, returned NULL object
    ``SingleExecutionState.ERROR``: error during iteration
    ``SingleExecutionState.ABORT``: iteration aborted
    ``SingleExecutionState.BUSY``: returned an element and iteration in progress	
    ``SingleExecutionState.IDLE``: ready for iteration

*)
METHOD iterate : CNM_ReturnTypes.SingleExecutionState
VAR_INPUT
	execute		:BOOL;
END_VAR
VAR_OUTPUT
	object 		:CNM_AbstractObject.IObject;
END_VAR
VAR_INST
	(*holds the state BUSY till the next cycle*)
	lastCycle	:BOOL;
	lastChangeVersion :__XWORD;
	cycleManager	:CNM_CycleManager.SimpleCycleManager;
END_VAR
VAR CONSTANT
	NULL :__XWORD := 0;
	INIT :DINT := CNM_ReturnTypes.DefaultSteps.STEP.INIT;
	ERROR :DINT := CNM_ReturnTypes.DefaultSteps.STEP.ERROR;
	SUCCESS :DINT := CNM_ReturnTypes.DefaultSteps.STEP.SUCCESS;
	ITERATING :DINT := INIT + 1;
END_VAR
cycleManager(execute := execute);
object := NULL;
CASE cycleManager.step.current OF
INIT:
	lastChangeVersion := THIS^.list.listChangeIndex;
	cycleManager.configuration.sequence.requireSuccessStep := FALSE;
	IF (THIS^.list.size = 0) THEN
		cycleManager.proceedWith(SUCCESS);
	ELSE
		THIS^.currentElement := SEL(THIS^.direction = IterationDirection.BACKWARD, THIS^.list.head, THIS^.list.last);
		IF THIS^.isObjectValid(THIS^.currentElement) THEN
			object := THIS^.currentElement.object;
			THIS^.currentElement := SEL(THIS^.direction = IterationDirection.BACKWARD, THIS^.currentElement.next, THIS^.currentElement.previous);
			cycleManager.proceed();
		ELSE
			cycleManager.proceedWith(ERROR);
		END_IF
	END_IF;
ITERATING:
	IF lastChangeVersion <> THIS^.list.listChangeIndex THEN
		cycleManager.proceedWith(ERROR);
	ELSE
		IF (NOT THIS^.isObjectValid(THIS^.currentElement)) THEN
			cycleManager.proceedWith(SUCCESS);
		ELSIF (NOT THIS^.isObjectValid(THIS^.currentElement.object)) THEN
			cycleManager.proceedWith(ERROR);
		ELSE
			object := THIS^.currentElement.object;
			THIS^.currentElement := SEL(THIS^.direction = IterationDirection.BACKWARD, THIS^.currentElement.next, THIS^.currentElement.previous);
		END_IF
	END_IF
END_CASE

THIS^.currentObject := object;
iterate := cycleManager.state;
END_METHOD

(*

## Short summary

This method resets the iterator.

**Example:**
```
iterator.reset();
WHILE(iterator.moveNext())DO
	foo := iterator.current.hashCode;
	bar := iterator.current.name;
END_WHILE
```

.. <legal notes>

legal notes
=================
| SPDX-FileCopyrightText: © 2022 ekvip automation GmbH <info@ekvip.de>
| SPDX-License-Identifier: Apache-2.0
| For details check: Apache-2.0_

.. _Apache-2.0: https://www.apache.org/licenses/LICENSE-2.0

.. </legal notes>

*)
METHOD reset
VAR CONSTANT
	NULL :__XWORD := 0; 
END_VAR
IF THIS^.isObjectValid(THIS^.list) THEN
	THIS^.currentElement := SEL(THIS^.direction = IterationDirection.BACKWARD, list.head, list.last);
END_IF
THIS^.iterate(FALSE);
THIS^.currentObject := NULL;
END_METHOD

END_FUNCTION_BLOCK

// ---- Lists/LinkedList/LinkedListSorter/LinkedListMergeSorter.TcPOU
(*

## Short summary

Implementation of an Inplace Mergesorter for the LinkedList

.. <legal notes>

legal notes
=================
| SPDX-FileCopyrightText: © 2025 ekvip automation GmbH <info@ekvip.de>
| SPDX-License-Identifier: Apache-2.0
| For details check: Apache-2.0_

.. _Apache-2.0: https://www.apache.org/licenses/LICENSE-2.0

.. </legal notes>



*)

{attribute 'enable_dynamic_creation'}
FUNCTION_BLOCK LinkedListMergeSorter EXTENDS AbstractLinkedListSorter

(*

## Short summary

This abstract property returns the class name of the concrete object, 
which is useful to check the class name for ``__DELETE``.

.. <legal notes>

legal notes
=================
| SPDX-FileCopyrightText: © 2022 ekvip automation GmbH <info@ekvip.de>
| SPDX-License-Identifier: Apache-2.0
| For details check: Apache-2.0_

.. _Apache-2.0: https://www.apache.org/licenses/LICENSE-2.0

.. </legal notes>

*)
PROPERTY className : CNM_AbstractObject.ClassName
GET
className := 'CNM_Collections.LinkedListMergeSorter';
END_GET
END_PROPERTY

(*

## Short summary

This method is used to create a new instance
of the object which has the same internal state as the object.
If the object is a container class, the references to the content objects
are not cloned for this there is the method `ICloneable.deepClone`.

If an object does not support cloning the return value is
``CNM_ReturnTypes.CloneResult.CLONE_IS_NOT_SUPPORTED``.

If there is not enough memory or the cloning fails because the
attribute enable dynamic creation was forgotten the return value is 
``CNM_ReturnTypes.CloneResult.FAILED``.

Only if the return value is ``CNM_ReturnTypes.CloneResult.SUCCESS``
the output ``clonedObject`` points to the new object
otherwise ``clonedObject`` is NULL.  

.. <legal notes>

legal notes
=================
| SPDX-FileCopyrightText: © 2022 ekvip automation GmbH <info@ekvip.de>
| SPDX-License-Identifier: Apache-2.0
| For details check: Apache-2.0_

.. _Apache-2.0: https://www.apache.org/licenses/LICENSE-2.0

.. </legal notes>


**Return:**``CNM_ReturnTypes.CloneResult.SUCCESS``: new object clone was created,
``CNM_ReturnTypes.CloneResult.FAILED``: object clone failed
``CNM_ReturnTypes.CloneResult.CLONE_IS_NOT_SUPPORTED``: object does not support cloning

*)
METHOD clone : CNM_AbstractObject.CNM_ReturnTypes.CloneResult
VAR
	newSorter :POINTER TO LinkedListMergeSorter;
END_VAR
VAR_OUTPUT
	(* new object instance or NULL if somthing went wrong *)
	clonedObject	: CNM_AbstractObject.IObject;
END_VAR
newSorter := __NEW(
	LinkedListMergeSorter()
);

IF (newSorter = 0) THEN
	clone := CNM_ReturnTypes.CloneResult.FAILED;
ELSE
	clone := CNM_ReturnTypes.CloneResult.SUCCESS;
	THIS^.prepareClonedSorter(newSorter^);
	clonedObject := newSorter^;
END_IF
END_METHOD

(*

## Short summary

This method sorts the data structure instantly within one call. 
Uses the passed Comparator or the compareTo of the contained Objects if no comparator is passed.

.. <legal notes>

legal notes
=================
| SPDX-FileCopyrightText: © 2022 ekvip automation GmbH <info@ekvip.de>
| SPDX-License-Identifier: Apache-2.0
| For details check: Apache-2.0_

.. _Apache-2.0: https://www.apache.org/licenses/LICENSE-2.0

.. </legal notes>


**Return:**``ERROR``: Sort was not able to finish 
	``SUCCESS``: Sorting was finished succesfully

